C07270=1013.905,188.212,370.193,167.076,55.174,160.197
C07271=1013.901,187.964,370.214,167.071,55.186,160.199
C07272=1013.897,187.715,370.234,167.066,55.198,160.200
C07273=1013.892,187.466,370.256,167.063,55.210,160.202
C07274=1013.889,187.217,370.278,167.058,55.222,160.203
C07275=1013.885,186.938,370.301,167.053,55.235,160.205
C07276=1013.881,186.658,370.325,167.049,55.249,160.206
C07277=1013.875,186.380,370.348,167.043,55.262,160.208
C07278=1013.871,186.100,370.372,167.039,55.275,160.209
C07279=1013.867,185.851,370.393,167.035,55.287,160.211
C07280=1013.863,185.602,370.414,167.030,55.299,160.212
C07281=1013.859,185.352,370.435,167.026,55.311,160.214
C07282=1013.855,185.104,370.456,167.023,55.323,160.215
C07283=1013.852,184.855,370.477,167.018,55.335,160.217
C07284=1013.847,184.605,370.499,167.013,55.347,160.218
C07285=1013.843,184.356,370.519,167.010,55.358,160.220
C07286=1013.839,184.108,370.540,167.005,55.370,160.221
C07287=1013.836,183.858,370.562,167.001,55.382,160.222
C07288=1013.832,183.609,370.583,166.997,55.393,160.224
C07289=1013.828,183.360,370.603,166.993,55.406,160.225
C07290=1013.824,183.110,370.624,166.989,55.418,160.227
C07291=1013.820,182.861,370.645,166.985,55.430,160.228
C07292=1013.817,182.613,370.666,166.980,55.441,160.230
C07293=1013.813,182.364,370.687,166.976,55.453,160.231
C07294=1013.809,182.114,370.708,166.972,55.465,160.233
C07295=1013.805,181.865,370.729,166.968,55.476,160.234
C07296=1013.801,181.615,370.750,166.964,55.488,160.235
C07297=1013.797,181.367,370.770,166.960,55.501,160.237
C07298=1013.793,181.118,370.791,166.956,55.512,160.239
C07299=1013.788,180.868,370.811,166.951,55.524,160.240
C07300=1013.784,180.619,370.832,166.947,55.537,160.241
C07301=1013.780,180.370,370.852,166.943,55.549,160.243
C07302=1013.776,180.122,370.872,166.939,55.561,160.244
C07303=1013.772,179.872,370.893,166.935,55.573,160.246
C07304=1013.767,179.623,370.912,166.931,55.585,160.247
C07305=1013.763,179.374,370.933,166.927,55.598,160.249
C07306=1013.760,179.124,370.953,166.923,55.609,160.250
C07307=1013.754,178.875,370.973,166.918,55.621,160.252
C07308=1013.751,178.626,370.994,166.914,55.634,160.253
C07309=1013.746,178.377,371.013,166.911,55.645,160.255
C07310=1013.743,178.128,371.034,166.906,55.657,160.256
C07311=1013.738,177.878,371.054,166.902,55.670,160.258
C07312=1013.734,177.630,371.074,166.898,55.682,160.259
C07313=1013.730,177.380,371.094,166.894,55.694,160.261
C07314=1013.726,177.131,371.114,166.890,55.706,160.262
C07315=1013.721,176.882,371.135,166.886,55.718,160.264
C07316=1013.718,176.633,371.155,166.882,55.730,160.265
C07317=1013.713,176.384,371.175,166.878,55.743,160.267
C07318=1013.709,176.135,371.195,166.875,55.754,160.268
C07319=1013.705,175.886,371.215,166.870,55.766,160.270
C07320=1013.701,175.636,371.235,166.866,55.778,160.271
C07321=1013.697,175.387,371.256,166.863,55.790,160.273
C07322=1013.693,175.138,371.276,166.858,55.802,160.274
C07323=1013.689,174.889,371.296,166.854,55.814,160.276
C07324=1013.685,174.640,371.315,166.851,55.827,160.278
C07325=1013.681,174.391,371.336,166.846,55.839,160.279
C07326=1013.677,174.141,371.356,166.843,55.850,160.280
C07327=1013.673,173.892,371.375,166.838,55.862,160.282
C07328=1013.668,173.642,371.396,166.835,55.875,160.284
C07329=1013.664,173.394,371.416,166.831,55.887,160.285
C07330=1013.660,173.145,371.436,166.826,55.899,160.286
C07331=1013.657,172.895,371.456,166.823,55.910,160.288
C07332=1013.652,172.646,371.476,166.819,55.923,160.289
C07333=1013.648,172.397,371.496,166.816,55.935,160.291
C07334=1013.644,172.148,371.516,166.811,55.947,160.292
C07335=1013.640,171.899,371.536,166.808,55.958,160.294
C07336=1013.636,171.650,371.555,166.803,55.970,160.295
C07337=1013.632,171.401,371.576,166.800,55.983,160.297
C07338=1013.629,171.151,371.596,166.796,55.995,160.298
C07339=1013.624,170.872,371.619,166.792,56.007,160.300
C07340=1013.619,170.593,371.641,166.787,56.021,160.302
C07341=1013.615,170.314,371.663,166.784,56.034,160.303
C07342=1013.610,170.034,371.685,166.779,56.048,160.305
C07343=1013.606,169.785,371.705,166.775,56.060,160.307
C07344=1013.603,169.536,371.725,166.771,56.072,160.308
C07345=1013.598,169.287,371.745,166.768,56.083,160.310
C07346=1013.595,169.037,371.765,166.763,56.095,160.311
C07347=1013.591,168.788,371.784,166.761,56.108,160.313
C07348=1013.587,168.539,371.804,166.756,56.120,160.314
C07349=1013.583,168.290,371.824,166.753,56.131,160.316
C07350=1013.579,168.041,371.845,166.749,56.143,160.317
C07351=1013.575,167.792,371.865,166.745,56.155,160.319
C07352=1013.571,167.543,371.884,166.742,56.167,160.320
C07353=1013.567,167.293,371.904,166.737,56.179,160.322
C07354=1013.563,167.044,371.924,166.734,56.190,160.323
C07355=1013.559,166.795,371.944,166.730,56.202,160.325
C07356=1013.556,166.546,371.964,166.726,56.214,160.326
C07357=1013.551,166.297,371.983,166.723,56.227,160.328
C07358=1013.548,166.047,372.003,166.720,56.238,160.329
C07359=1013.543,165.798,372.023,166.715,56.250,160.331
C07360=1013.540,165.549,372.043,166.712,56.262,160.332
C07361=1013.535,165.300,372.062,166.709,56.274,160.334
C07362=1013.532,165.050,372.082,166.704,56.286,160.335
C07363=1013.528,164.801,372.102,166.701,56.297,160.337
C07364=1013.524,164.552,372.122,166.698,56.309,160.338
C07365=1013.521,164.303,372.142,166.694,56.321,160.340
C07366=1013.517,164.054,372.160,166.690,56.333,160.341
C07367=1013.513,163.804,372.180,166.687,56.345,160.343
C07368=1013.509,163.555,372.200,166.683,56.356,160.344
C07369=1013.505,163.306,372.220,166.680,56.368,160.346
C07370=1013.501,163.057,372.240,166.676,56.380,160.347
C07371=1013.497,162.808,372.259,166.672,56.392,160.349
C07372=1013.493,162.558,372.280,166.669,56.403,160.350
C07373=1013.490,162.310,372.299,166.666,56.415,160.352
C07374=1013.486,162.061,372.319,166.661,56.427,160.353
C07375=1013.482,161.812,372.338,166.658,56.439,160.355
C07376=1013.478,161.562,372.358,166.654,56.450,160.356
C07377=1013.475,161.312,372.378,166.651,56.462,160.358
C07378=1013.471,161.063,372.397,166.648,56.473,160.359
C07379=1013.467,160.814,372.417,166.644,56.485,160.361
C07380=1013.463,160.565,372.436,166.640,56.497,160.362
C07381=1013.460,160.316,372.456,166.637,56.509,160.364
C07382=1013.456,160.066,372.476,166.633,56.521,160.365
C07383=1013.452,159.817,372.495,166.630,56.532,160.367
C07384=1013.448,159.568,372.515,166.627,56.544,160.368
C07385=1013.445,159.319,372.534,166.624,56.556,160.370
C07386=1013.441,159.070,372.554,166.620,56.567,160.371
C07387=1013.437,158.820,372.573,166.616,56.579,160.373
C07388=1013.433,158.571,372.593,166.612,56.591,160.374
C07389=1013.430,158.322,372.613,166.609,56.603,160.376
C07390=1013.426,158.072,372.632,166.606,56.614,160.377
C07391=1013.421,157.823,372.652,166.603,56.626,160.379
C07392=1013.418,157.574,372.670,166.599,56.638,160.381
C07393=1013.413,157.325,372.689,166.595,56.650,160.382
C07394=1013.410,157.075,372.709,166.592,56.662,160.384
C07395=1013.406,156.826,372.728,166.589,56.673,160.385
C07396=1013.402,156.577,372.747,166.585,56.685,160.387
C07397=1013.398,156.328,372.766,166.582,56.697,160.388
C07398=1013.394,156.078,372.785,166.578,56.709,160.390
C07399=1013.390,155.829,372.804,166.575,56.721,160.391
C07400=1013.386,155.580,372.823,166.571,56.733,160.393
C07401=1013.382,155.331,372.842,166.568,56.744,160.394
C07402=1013.378,155.082,372.861,166.565,56.756,160.396
C07403=1013.374,154.802,372.882,166.560,56.769,160.397
C07404=1013.370,154.522,372.904,166.557,56.783,160.399
C07405=1013.365,154.243,372.925,166.553,56.796,160.401
C07406=1013.360,153.963,372.947,166.550,56.809,160.403
C07407=1013.357,153.714,372.965,166.547,56.821,160.404
C07408=1013.352,153.465,372.984,166.542,56.833,160.406
C07409=1013.348,153.216,373.003,166.539,56.845,160.407
C07410=1013.344,152.966,373.022,166.536,56.857,160.409
C07411=1013.341,152.718,373.041,166.533,56.868,160.411
C07412=1013.337,152.468,373.060,166.530,56.880,160.412
C07413=1013.333,152.218,373.079,166.526,56.891,160.413
C07414=1013.329,151.970,373.098,166.523,56.903,160.415
C07415=1013.325,151.720,373.116,166.520,56.915,160.417
C07416=1013.321,151.471,373.135,166.516,56.927,160.418
C07417=1013.317,151.222,373.154,166.513,56.938,160.420
C07418=1013.313,150.972,373.172,166.510,56.950,160.421
C07419=1013.309,150.723,373.192,166.507,56.962,160.423
C07420=1013.305,150.474,373.210,166.503,56.974,160.424
C07421=1013.301,150.224,373.229,166.500,56.986,160.426
C07422=1013.297,149.975,373.248,166.497,56.998,160.427
C07423=1013.293,149.726,373.267,166.493,57.009,160.429
C07424=1013.289,149.477,373.286,166.490,57.021,160.430
C07425=1013.285,149.227,373.304,166.487,57.033,160.432
C07426=1013.282,148.978,373.323,166.483,57.044,160.434
C07427=1013.278,148.728,373.341,166.480,57.056,160.435
C07428=1013.274,148.479,373.360,166.477,57.068,160.437
C07429=1013.270,148.230,373.379,166.474,57.079,160.438
C07430=1013.266,147.981,373.398,166.470,57.091,160.440
C07431=1013.262,147.732,373.416,166.467,57.103,160.441
C07432=1013.258,147.482,373.435,166.464,57.115,160.443
C07433=1013.254,147.233,373.453,166.461,57.126,160.444
C07434=1013.250,146.984,373.472,166.457,57.138,160.446
C07435=1013.246,146.734,373.491,166.454,57.149,160.447
C07436=1013.243,146.485,373.509,166.451,57.161,160.449
C07437=1013.239,146.235,373.528,166.449,57.173,160.451
C07438=1013.235,145.987,373.545,166.446,57.184,160.452
C07439=1013.231,145.737,373.564,166.442,57.196,160.454
C07440=1013.227,145.487,373.583,166.439,57.207,160.455
C07441=1013.223,145.239,373.602,166.436,57.219,160.457
C07442=1013.219,144.989,373.621,166.433,57.231,160.458
C07443=1013.215,144.740,373.638,166.430,57.242,160.460
C07444=1013.211,144.491,373.657,166.427,57.254,160.461
C07445=1013.207,144.242,373.675,166.424,57.266,160.463
C07446=1013.203,143.992,373.693,166.420,57.278,160.465
C07447=1013.199,143.743,373.712,166.417,57.290,160.466
C07448=1013.195,143.494,373.730,166.414,57.301,160.468
C07449=1013.191,143.245,373.748,166.411,57.313,160.469
C07450=1013.187,142.995,373.767,166.408,57.325,160.471
C07451=1013.183,142.746,373.786,166.405,57.336,160.472
C07452=1013.179,142.496,373.803,166.402,57.347,160.474
C07453=1013.175,142.247,373.822,166.399,57.359,160.475
C07454=1013.172,141.998,373.840,166.396,57.371,160.477
C07455=1013.167,141.748,373.858,166.392,57.382,160.478
C07456=1013.163,141.499,373.876,166.389,57.394,160.480
C07457=1013.159,141.250,373.895,166.386,57.406,160.482
C07458=1013.155,141.000,373.912,166.383,57.417,160.483
C07459=1013.152,140.752,373.931,166.381,57.428,160.485
C07460=1013.148,140.502,373.949,166.378,57.440,160.486
C07461=1013.144,140.253,373.967,166.374,57.452,160.488
C07462=1013.140,140.004,373.986,166.371,57.463,160.489
C07463=1013.136,139.754,374.003,166.368,57.475,160.491
C07464=1013.132,139.505,374.022,166.366,57.486,160.492
C07465=1013.128,139.256,374.040,166.363,57.498,160.494
C07466=1013.124,139.006,374.058,166.359,57.509,160.495
C07467=1013.120,138.726,374.079,166.356,57.522,160.497
C07468=1013.115,138.447,374.100,166.352,57.535,160.499
C07469=1013.111,138.167,374.119,166.350,57.548,160.501
C07470=1013.107,137.888,374.140,166.347,57.561,160.503
C07471=1013.103,137.639,374.158,166.343,57.572,160.504
C07472=1013.099,137.389,374.176,166.340,57.584,160.506
C07473=1013.095,137.140,374.194,166.338,57.595,160.507
C07474=1013.090,136.891,374.212,166.335,57.607,160.509
C07475=1013.087,136.641,374.230,166.332,57.619,160.510
C07476=1013.083,136.393,374.248,166.328,57.630,160.512
C07477=1013.079,136.142,374.266,166.326,57.641,160.513
C07478=1013.075,135.894,374.284,166.323,57.653,160.515
C07479=1013.071,135.644,374.302,166.320,57.665,160.516
C07480=1013.067,135.395,374.320,166.316,57.676,160.518
C07481=1013.064,135.146,374.338,166.314,57.687,160.520
C07482=1013.059,134.896,374.355,166.311,57.698,160.521
C07483=1013.055,134.647,374.373,166.308,57.710,160.523
C07484=1013.051,134.397,374.391,166.305,57.721,160.524
C07485=1013.047,134.148,374.409,166.302,57.733,160.526
C07486=1013.044,133.899,374.427,166.299,57.744,160.527
C07487=1013.039,133.649,374.445,166.297,57.756,160.529
C07488=1013.035,133.400,374.462,166.294,57.767,160.530
C07489=1013.032,133.151,374.480,166.291,57.779,160.532
C07490=1013.028,132.901,374.498,166.288,57.790,160.533
C07491=1013.023,132.653,374.516,166.285,57.802,160.535
C07492=1013.020,132.403,374.533,166.282,57.813,160.536
C07493=1013.015,132.154,374.551,166.279,57.824,160.538
C07494=1013.012,131.904,374.569,166.277,57.836,160.540
C07495=1013.008,131.655,374.587,166.274,57.847,160.541
C07496=1013.004,131.405,374.604,166.271,57.859,160.543
C07497=1013.001,131.156,374.622,166.268,57.870,160.544
C07498=1012.996,130.907,374.640,166.265,57.881,160.546
C07499=1012.992,130.657,374.657,166.263,57.893,160.547
C07500=1012.988,130.408,374.676,166.260,57.903,160.549
C07501=1012.985,130.159,374.693,166.257,57.915,160.550
C07502=1012.981,129.909,374.711,166.255,57.926,160.552
C07503=1012.977,129.660,374.729,166.251,57.937,160.553
C07504=1012.973,129.411,374.746,166.249,57.948,160.555
C07505=1012.969,129.161,374.764,166.246,57.960,160.557
C07506=1012.965,128.912,374.781,166.243,57.972,160.558
C07507=1012.961,128.663,374.799,166.240,57.982,160.559
C07508=1012.957,128.413,374.816,166.237,57.994,160.561
C07509=1012.953,128.163,374.833,166.235,58.005,160.563
C07510=1012.949,127.914,374.850,166.232,58.017,160.564
C07511=1012.945,127.665,374.868,166.229,58.028,160.566
C07512=1012.940,127.415,374.885,166.226,58.039,160.567
C07513=1012.936,127.166,374.902,166.224,58.051,160.569
C07514=1012.932,126.917,374.920,166.221,58.062,160.570
C07515=1012.928,126.667,374.937,166.218,58.073,160.572
C07516=1012.924,126.418,374.954,166.216,58.085,160.574
C07517=1012.920,126.168,374.971,166.213,58.096,160.575
C07518=1012.916,125.920,374.989,166.210,58.107,160.577
C07519=1012.911,125.670,375.006,166.208,58.119,160.578
C07520=1012.908,125.420,375.023,166.205,58.130,160.580
C07521=1012.904,125.171,375.041,166.202,58.141,160.581
C07522=1012.900,124.922,375.058,166.199,58.152,160.583
C07523=1012.896,124.673,375.075,166.197,58.164,160.584
C07524=1012.892,124.423,375.092,166.194,58.175,160.586
C07525=1012.888,124.173,375.109,166.191,58.186,160.587
C07526=1012.884,123.924,375.126,166.189,58.197,160.589
C07527=1012.880,123.675,375.143,166.186,58.208,160.591
C07528=1012.876,123.426,375.161,166.184,58.220,160.592
C07529=1012.871,123.176,375.179,166.181,58.231,160.594
C07530=1012.867,122.927,375.196,166.178,58.242,160.595
C07531=1012.863,122.621,375.216,166.175,58.255,160.597
C07532=1012.858,122.316,375.237,166.172,58.269,160.599
C07533=1012.853,122.010,375.258,166.169,58.282,160.601
C07534=1012.849,121.705,375.280,166.165,58.296,160.602
C07535=1012.844,121.455,375.297,166.162,58.307,160.604
C07536=1012.840,121.206,375.314,166.160,58.318,160.606
C07537=1012.836,120.956,375.331,166.158,58.330,160.607
C07538=1012.832,120.707,375.348,166.155,58.341,160.609
C07539=1012.829,120.458,375.366,166.153,58.352,160.610
C07540=1012.825,120.208,375.383,166.151,58.363,160.612
C07541=1012.820,119.959,375.400,166.147,58.374,160.613
C07542=1012.816,119.709,375.417,166.145,58.385,160.615
C07543=1012.813,119.460,375.434,166.142,58.395,160.616
C07544=1012.809,119.211,375.451,166.140,58.406,160.618
C07545=1012.805,118.961,375.468,166.136,58.417,160.619
C07546=1012.801,118.712,375.485,166.134,58.428,160.621
C07547=1012.797,118.463,375.503,166.132,58.439,160.622
C07548=1012.793,118.214,375.520,166.130,58.450,160.624
C07549=1012.789,117.964,375.537,166.127,58.461,160.626
C07550=1012.785,117.714,375.554,166.124,58.472,160.627
C07551=1012.781,117.465,375.571,166.122,58.483,160.628
C07552=1012.777,117.216,375.588,166.120,58.494,160.630
C07553=1012.773,116.966,375.605,166.117,58.504,160.631
C07554=1012.770,116.717,375.622,166.115,58.515,160.633
C07555=1012.766,116.467,375.639,166.112,58.526,160.635
C07556=1012.762,116.218,375.656,166.110,58.537,160.636
C07557=1012.758,115.969,375.673,166.108,58.548,160.638
C07558=1012.754,115.720,375.690,166.104,58.558,160.639
C07559=1012.750,115.470,375.707,166.102,58.569,160.640
C07560=1012.746,115.221,375.724,166.099,58.580,160.642
C07561=1012.742,114.971,375.742,166.097,58.591,160.644
C07562=1012.738,114.722,375.759,166.094,58.601,160.645
C07563=1012.734,114.472,375.775,166.092,58.612,160.646
C07564=1012.731,114.223,375.792,166.090,58.623,160.648
C07565=1012.727,113.973,375.809,166.087,58.633,160.649
C07566=1012.723,113.724,375.826,166.085,58.644,160.651
C07567=1012.719,113.475,375.843,166.083,58.655,160.652
C07568=1012.715,113.226,375.860,166.080,58.665,160.654
C07569=1012.711,112.976,375.878,166.078,58.676,160.655
C07570=1012.708,112.726,375.894,166.076,58.687,160.657
C07571=1012.704,112.477,375.911,166.073,58.697,160.658
C07572=1012.700,112.228,375.928,166.071,58.708,160.660
C07573=1012.696,111.979,375.945,166.068,58.719,160.661
C07574=1012.692,111.729,375.962,166.066,58.729,160.663
C07575=1012.689,111.479,375.979,166.063,58.740,160.664
C07576=1012.685,111.230,375.996,166.061,58.751,160.666
C07577=1012.680,110.981,376.012,166.059,58.762,160.667
C07578=1012.677,110.731,376.029,166.056,58.772,160.669
C07579=1012.673,110.482,376.046,166.054,58.783,160.670
C07580=1012.669,110.233,376.063,166.051,58.794,160.672
C07581=1012.664,109.983,376.078,166.050,58.803,160.673
C07582=1012.661,109.734,376.096,166.048,58.814,160.675
C07583=1012.657,109.484,376.112,166.045,58.825,160.676
C07584=1012.652,109.235,376.128,166.043,58.836,160.678
C07585=1012.649,108.986,376.145,166.040,58.846,160.679
C07586=1012.645,108.736,376.162,166.038,58.857,160.681
C07587=1012.611,121.701,374.880,166.126,58.488,160.631
C07588=1012.616,121.999,374.859,166.130,58.476,160.629
C07589=1012.621,122.296,374.839,166.133,58.462,160.627
C07590=1012.625,122.594,374.819,166.135,58.450,160.625
C07591=1012.629,122.892,374.799,166.138,58.436,160.624
C07592=1012.634,123.142,374.781,166.142,58.425,160.622
C07593=1012.638,123.391,374.764,166.144,58.414,160.621
C07594=1012.642,123.640,374.747,166.146,58.403,160.619
C07595=1012.646,123.890,374.730,166.148,58.392,160.617
C07596=1012.649,124.139,374.713,166.152,58.381,160.616
C07597=1012.653,124.388,374.696,166.154,58.370,160.615
C07598=1012.657,124.637,374.679,166.157,58.359,160.613
C07599=1012.662,124.887,374.661,166.160,58.348,160.612
C07600=1012.666,125.137,374.644,166.162,58.337,160.610
C07601=1012.669,125.386,374.627,166.165,58.326,160.609
C07602=1012.673,125.635,374.610,166.167,58.314,160.607
C07603=1012.677,125.884,374.593,166.169,58.303,160.605
C07604=1012.682,126.134,374.575,166.173,58.292,160.604
C07605=1012.686,126.383,374.558,166.175,58.281,160.602
C07606=1012.690,126.632,374.541,166.178,58.270,160.601
C07607=1012.694,126.882,374.523,166.181,58.259,160.599
C07608=1012.697,127.131,374.506,166.183,58.247,160.598
C07609=1012.702,127.381,374.489,166.186,58.236,160.596
C07610=1012.706,127.630,374.472,166.189,58.225,160.595
C07611=1012.710,127.879,374.455,166.191,58.214,160.593
C07612=1012.714,128.129,374.438,166.195,58.202,160.592
C07613=1012.717,128.378,374.421,166.196,58.191,160.590
C07614=1012.722,128.628,374.403,166.200,58.180,160.588
C07615=1012.726,128.877,374.386,166.202,58.169,160.587
C07616=1012.730,129.126,374.369,166.205,58.157,160.586
C07617=1012.734,129.375,374.351,166.207,58.146,160.584
C07618=1012.738,129.625,374.333,166.211,58.135,160.582
C07619=1012.741,129.875,374.316,166.213,58.124,160.581
C07620=1012.745,130.124,374.298,166.216,58.112,160.579
C07621=1012.749,130.373,374.281,166.219,58.102,160.578
C07622=1012.753,130.623,374.263,166.222,58.090,160.576
C07623=1012.757,130.872,374.245,166.224,58.079,160.575
C07624=1012.760,131.121,374.228,166.227,58.067,160.573
C07625=1012.764,131.371,374.210,166.230,58.057,160.572
C07626=1012.768,131.620,374.192,166.232,58.045,160.570
C07627=1012.772,131.869,374.175,166.235,58.034,160.568
C07628=1012.775,132.119,374.157,166.238,58.023,160.567
C07629=1012.780,132.368,374.139,166.241,58.012,160.566
C07630=1012.784,132.617,374.122,166.243,58.000,160.564
C07631=1012.788,132.866,374.104,166.246,57.989,160.562
C07632=1012.791,133.116,374.086,166.249,57.978,160.561
C07633=1012.795,133.366,374.068,166.252,57.966,160.559
C07634=1012.799,133.615,374.051,166.255,57.955,160.558
C07635=1012.803,133.864,374.034,166.258,57.944,160.556
C07636=1012.807,134.114,374.015,166.260,57.932,160.555
C07637=1012.811,134.363,373.998,166.263,57.921,160.553
C07638=1012.815,134.612,373.981,166.266,57.909,160.552
C07639=1012.819,134.862,373.962,166.268,57.898,160.550
C07640=1012.823,135.111,373.945,166.272,57.887,160.549
C07641=1012.826,135.360,373.926,166.275,57.875,160.547
C07642=1012.831,135.610,373.909,166.277,57.864,160.546
C07643=1012.834,135.859,373.891,166.280,57.852,160.544
C07644=1012.838,136.108,373.873,166.284,57.841,160.543
C07645=1012.842,136.358,373.855,166.285,57.829,160.541
C07646=1012.846,136.607,373.838,166.289,57.818,160.539
C07647=1012.849,136.856,373.819,166.292,57.807,160.538
C07648=1012.854,137.105,373.801,166.294,57.795,160.536
C07649=1012.857,137.355,373.783,166.298,57.784,160.535
C07650=1012.862,137.604,373.766,166.301,57.772,160.533
C07651=1012.865,137.854,373.748,166.303,57.761,160.532
C07652=1012.870,138.133,373.727,166.306,57.748,160.530
C07653=1012.874,138.413,373.707,166.310,57.735,160.528
C07654=1012.878,138.691,373.687,166.314,57.723,160.527
C07655=1012.882,138.971,373.667,166.316,57.710,160.525
C07656=1012.887,139.221,373.648,166.319,57.698,160.523
C07657=1012.890,139.470,373.630,166.322,57.687,160.522
C07658=1012.894,139.719,373.613,166.325,57.675,160.520
C07659=1012.898,139.969,373.594,166.328,57.664,160.519
C07660=1012.902,140.217,373.576,166.331,57.652,160.517
C07661=1012.906,140.467,373.557,166.334,57.641,160.516
C07662=1012.909,140.717,373.540,166.337,57.629,160.514
C07663=1012.914,140.966,373.522,166.341,57.618,160.513
C07664=1012.917,141.215,373.503,166.343,57.606,160.511
C07665=1012.921,141.464,373.485,166.346,57.594,160.509
C07666=1012.925,141.714,373.467,166.349,57.583,160.508
C07667=1012.929,141.963,373.449,166.352,57.571,160.506
C07668=1012.933,142.212,373.430,166.356,57.560,160.505
C07669=1012.937,142.461,373.412,166.359,57.548,160.503
C07670=1012.941,142.711,373.394,166.361,57.537,160.501
C07671=1012.944,142.960,373.376,166.364,57.526,160.500
C07672=1012.949,143.210,373.358,166.367,57.514,160.498
C07673=1012.952,143.459,373.339,166.370,57.502,160.497
C07674=1012.956,143.708,373.321,166.374,57.491,160.496
C07675=1012.960,143.958,373.304,166.377,57.479,160.494
C07676=1012.964,144.206,373.285,166.380,57.467,160.492
C07677=1012.968,144.456,373.266,166.383,57.455,160.491
C07678=1012.972,144.705,373.249,166.386,57.444,160.489
C07679=1012.976,144.954,373.230,166.389,57.432,160.488
C07680=1012.979,145.203,373.211,166.392,57.420,160.486
C07681=1012.984,145.453,373.193,166.395,57.409,160.485
C07682=1012.987,145.702,373.176,166.398,57.397,160.483
C07683=1012.991,145.952,373.157,166.401,57.385,160.481
C07684=1012.995,146.202,373.138,166.404,57.374,160.480
C07685=1012.999,146.451,373.120,166.407,57.362,160.478
C07686=1013.003,146.700,373.101,166.410,57.351,160.477
C07687=1013.006,146.949,373.083,166.414,57.339,160.475
C07688=1013.010,147.199,373.064,166.417,57.327,160.474
C07689=1013.015,147.448,373.046,166.420,57.316,160.472
C07690=1013.019,147.697,373.027,166.423,57.304,160.471
C07691=1013.022,147.946,373.009,166.426,57.292,160.469
C07692=1013.026,148.196,372.990,166.430,57.281,160.468
C07693=1013.030,148.444,372.971,166.433,57.269,160.466
C07694=1013.034,148.694,372.952,166.436,57.257,160.464
C07695=1013.038,148.943,372.934,166.439,57.245,160.463
C07696=1013.041,149.192,372.915,166.443,57.234,160.462
C07697=1013.045,149.442,372.896,166.446,57.222,160.460
C07698=1013.049,149.691,372.878,166.449,57.210,160.458
C07699=1013.053,149.941,372.859,166.452,57.198,160.457
C07700=1013.056,150.190,372.841,166.455,57.187,160.455
C07701=1013.060,150.439,372.822,166.459,57.176,160.454
C07702=1013.065,150.688,372.803,166.462,57.164,160.452
C07703=1013.069,150.937,372.785,166.465,57.152,160.451
C07704=1013.073,151.187,372.766,166.468,57.140,160.449
C07705=1013.076,151.436,372.748,166.471,57.128,160.447
C07706=1013.081,151.685,372.729,166.474,57.116,160.446
C07707=1013.085,151.935,372.710,166.477,57.104,160.444
C07708=1013.088,152.184,372.692,166.482,57.093,160.443
C07709=1013.092,152.433,372.672,166.485,57.081,160.441
C07710=1013.096,152.683,372.654,166.488,57.069,160.440
C07711=1013.100,152.932,372.635,166.491,57.057,160.438
C07712=1013.104,153.181,372.616,166.494,57.046,160.437
C07713=1013.107,153.430,372.597,166.497,57.034,160.435
C07714=1013.111,153.680,372.578,166.501,57.022,160.434
C07715=1013.115,153.929,372.559,166.504,57.011,160.432
C07716=1013.120,154.208,372.538,166.507,56.997,160.430
C07717=1013.124,154.487,372.517,166.512,56.984,160.429
C07718=1013.128,154.767,372.495,166.516,56.971,160.427
C07719=1013.133,155.047,372.474,166.519,56.958,160.425
C07720=1013.137,155.295,372.455,166.522,56.946,160.424
C07721=1013.141,155.545,372.437,166.527,56.934,160.422
C07722=1013.144,155.795,372.417,166.530,56.922,160.421
C07723=1013.148,156.043,372.398,166.533,56.910,160.419
C07724=1013.152,156.293,372.379,166.536,56.899,160.418
C07725=1013.156,156.542,372.361,166.539,56.887,160.416
C07726=1013.160,156.791,372.341,166.543,56.875,160.415
C07727=1013.163,157.040,372.323,166.547,56.863,160.413
C07728=1013.168,157.289,372.303,166.550,56.851,160.411
C07729=1013.172,157.539,372.285,166.553,56.839,160.410
C07730=1013.175,157.788,372.266,166.557,56.827,160.408
C07731=1013.180,158.037,372.247,166.560,56.815,160.407
C07732=1013.183,158.287,372.227,166.563,56.803,160.405
C07733=1013.187,158.536,372.208,166.567,56.792,160.404
C07734=1013.191,158.785,372.188,166.570,56.780,160.402
C07735=1013.194,159.035,372.169,166.573,56.768,160.400
C07736=1013.198,159.284,372.149,166.577,56.757,160.399
C07737=1013.202,159.533,372.129,166.581,56.745,160.398
C07738=1013.206,159.783,372.110,166.584,56.733,160.396
C07739=1013.209,160.031,372.091,166.588,56.721,160.395
C07740=1013.212,160.281,372.071,166.591,56.710,160.393
C07741=1013.217,160.530,372.051,166.594,56.698,160.391
C07742=1013.220,160.780,372.032,166.597,56.686,160.390
C07743=1013.224,161.028,372.013,166.601,56.674,160.389
C07744=1013.227,161.277,371.993,166.605,56.662,160.387
C07745=1013.232,161.526,371.973,166.608,56.651,160.386
C07746=1013.235,161.776,371.954,166.612,56.639,160.384
C07747=1013.239,162.026,371.934,166.615,56.628,160.383
C07748=1013.242,162.274,371.915,166.619,56.615,160.381
C07749=1013.246,162.523,371.895,166.622,56.604,160.380
C07750=1013.250,162.772,371.875,166.626,56.592,160.378
C07751=1013.254,163.022,371.856,166.629,56.580,160.376
C07752=1013.258,163.271,371.836,166.633,56.568,160.375
C07753=1013.261,163.520,371.817,166.637,56.556,160.373
C07754=1013.265,163.769,371.797,166.640,56.545,160.372
C07755=1013.269,164.019,371.777,166.644,56.533,160.371
C07756=1013.272,164.268,371.757,166.647,56.521,160.369
C07757=1013.277,164.517,371.738,166.651,56.509,160.367
C07758=1013.280,164.767,371.718,166.655,56.497,160.366
C07759=1013.283,165.016,371.699,166.658,56.485,160.364
C07760=1013.287,165.265,371.679,166.662,56.473,160.363
C07761=1013.291,165.514,371.659,166.666,56.461,160.361
C07762=1013.295,165.763,371.640,166.669,56.450,160.360
C07763=1013.299,166.012,371.619,166.672,56.438,160.358
C07764=1013.303,166.261,371.600,166.677,56.426,160.357
C07765=1013.307,166.511,371.580,166.680,56.414,160.355
C07766=1013.311,166.760,371.560,166.683,56.402,160.354
C07767=1013.315,167.009,371.540,166.687,56.390,160.352
C07768=1013.318,167.258,371.521,166.690,56.378,160.351
C07769=1013.322,167.507,371.502,166.695,56.366,160.349
C07770=1013.326,167.757,371.482,166.698,56.354,160.348
C07771=1013.329,168.006,371.462,166.701,56.342,160.346
C07772=1013.334,168.255,371.442,166.706,56.330,160.345
C07773=1013.337,168.505,371.422,166.709,56.319,160.343
C07774=1013.342,168.754,371.403,166.714,56.307,160.342
C07775=1013.345,169.003,371.383,166.716,56.294,160.340
C07776=1013.349,169.252,371.363,166.721,56.282,160.339
C07777=1013.353,169.501,371.343,166.724,56.270,160.337
C07778=1013.357,169.751,371.323,166.728,56.258,160.336
C07779=1013.361,170.000,371.304,166.732,56.247,160.334
C07780=1013.366,170.278,371.281,166.736,56.233,160.332
C07781=1013.370,170.557,371.259,166.740,56.220,160.331
C07782=1013.374,170.837,371.236,166.744,56.206,160.329
C07783=1013.379,171.116,371.214,166.749,56.193,160.327
C07784=1013.383,171.365,371.194,166.752,56.180,160.326
C07785=1013.386,171.615,371.174,166.756,56.168,160.324
C07786=1013.391,171.864,371.155,166.760,56.157,160.323
C07787=1013.394,172.113,371.135,166.764,56.145,160.321
C07788=1013.398,172.362,371.115,166.768,56.133,160.320
C07789=1013.402,172.611,371.095,166.772,56.120,160.318
C07790=1013.406,172.861,371.075,166.776,56.108,160.317
C07791=1013.411,173.109,371.055,166.779,56.096,160.315
C07792=1013.414,173.359,371.035,166.784,56.084,160.314
C07793=1013.418,173.608,371.015,166.787,56.072,160.312
C07794=1013.422,173.857,370.995,166.791,56.060,160.311
C07795=1013.426,174.106,370.975,166.796,56.048,160.309
C07796=1013.430,174.355,370.956,166.798,56.036,160.307
C07797=1013.434,174.604,370.935,166.803,56.024,160.306
C07798=1013.438,174.853,370.915,166.807,56.011,160.305
C07799=1013.443,175.103,370.895,166.811,56.000,160.303
C07800=1013.446,175.352,370.875,166.815,55.987,160.302
C07801=1013.451,175.602,370.856,166.818,55.976,160.300
C07802=1013.455,175.850,370.835,166.823,55.963,160.299
C07803=1013.458,176.100,370.815,166.826,55.951,160.297
C07804=1013.462,176.349,370.795,166.831,55.939,160.296
C07805=1013.466,176.598,370.775,166.834,55.927,160.294
C07806=1013.471,176.846,370.755,166.838,55.914,160.292
C07807=1013.474,177.096,370.735,166.843,55.902,160.291
C07808=1013.479,177.346,370.715,166.846,55.891,160.290
C07809=1013.483,177.595,370.695,166.850,55.878,160.288
C07810=1013.487,177.844,370.674,166.855,55.866,160.287
C07811=1013.491,178.093,370.655,166.859,55.853,160.285
C07812=1013.495,178.342,370.635,166.862,55.842,160.283
C07813=1013.499,178.590,370.615,166.867,55.830,160.282
C07814=1013.504,178.840,370.594,166.871,55.817,160.280
C07815=1013.507,179.090,370.574,166.875,55.805,160.279
C07816=1013.512,179.338,370.554,166.879,55.793,160.277
C07817=1013.516,179.588,370.534,166.883,55.781,160.276
C07818=1013.520,179.837,370.514,166.887,55.769,160.274
C07819=1013.524,180.086,370.493,166.891,55.756,160.273
C07820=1013.528,180.335,370.473,166.896,55.744,160.272
C07821=1013.532,180.584,370.454,166.899,55.732,160.270
C07822=1013.536,180.833,370.433,166.903,55.720,160.268
C07823=1013.541,181.082,370.413,166.908,55.708,160.267
C07824=1013.545,181.332,370.392,166.912,55.695,160.265
C07825=1013.549,181.581,370.372,166.916,55.683,160.264
C07826=1013.552,181.830,370.351,166.920,55.672,160.262
C07827=1013.556,182.080,370.330,166.924,55.660,160.261
C07828=1013.560,182.329,370.310,166.928,55.647,160.259
C07829=1013.564,182.578,370.289,166.932,55.635,160.258
C07830=1013.567,182.827,370.267,166.936,55.623,160.257
C07831=1013.572,183.076,370.246,166.941,55.612,160.255
C07832=1013.575,183.325,370.226,166.944,55.600,160.254
C07833=1013.579,183.574,370.206,166.949,55.588,160.252
C07834=1013.582,183.823,370.184,166.953,55.575,160.251
C07835=1013.587,184.073,370.163,166.957,55.564,160.249
C07836=1013.591,184.321,370.142,166.961,55.552,160.248
C07837=1013.595,184.570,370.121,166.966,55.540,160.247
C07838=1013.598,184.819,370.100,166.969,55.528,160.245
C07839=1013.602,185.069,370.080,166.973,55.516,160.243
C07840=1013.606,185.318,370.059,166.978,55.504,160.242
C07841=1013.610,185.567,370.038,166.983,55.492,160.241
C07842=1013.614,185.816,370.016,166.986,55.480,160.239
C07843=1013.618,186.065,369.996,166.990,55.468,160.238
C07844=1013.622,186.344,369.972,166.995,55.455,160.236
C07845=1013.626,186.624,369.948,167.000,55.441,160.234
C07846=1013.631,186.903,369.925,167.005,55.428,160.233
C07847=1013.635,187.182,369.901,167.010,55.414,160.231
C07848=1013.639,187.431,369.880,167.014,55.402,160.230
C07849=1013.643,187.680,369.860,167.019,55.390,160.228
C07850=1013.647,187.929,369.838,167.022,55.378,160.227
C07851=1013.651,188.178,369.817,167.027,55.366,160.225
C07852=1013.654,188.427,369.796,167.031,55.354,160.224
C07853=1013.659,188.676,369.775,167.035,55.342,160.222
C07854=1013.663,188.925,369.754,167.040,55.330,160.221
C07855=1013.667,189.175,369.733,167.045,55.318,160.220
C07856=1013.671,189.423,369.712,167.049,55.306,160.218
C07857=1013.674,189.672,369.691,167.052,55.294,160.217
C07858=1013.679,189.921,369.669,167.057,55.282,160.215
C07859=1013.682,190.170,369.648,167.062,55.270,160.214
C07860=1013.687,190.419,369.627,167.066,55.258,160.212
C07861=1013.691,190.668,369.606,167.071,55.246,160.211
C07862=1013.695,190.918,369.584,167.075,55.234,160.210
C07863=1013.699,191.167,369.563,167.079,55.221,160.208
C07864=1013.703,191.415,369.543,167.084,55.209,160.207
C07865=1013.707,191.665,369.521,167.089,55.197,160.205
C07866=1013.710,191.914,369.500,167.093,55.185,160.204
C07867=1013.715,192.163,369.479,167.098,55.173,160.202
C07868=1013.719,192.411,369.457,167.102,55.161,160.201
C07869=1013.723,192.661,369.436,167.105,55.149,160.199
C07870=1013.727,192.910,369.415,167.110,55.137,160.198
C07871=1013.731,193.159,369.394,167.115,55.125,160.196
C07872=1013.735,193.408,369.373,167.119,55.113,160.195
C07873=1013.739,193.657,369.350,167.124,55.101,160.194
C07874=1013.743,193.906,369.330,167.128,55.089,160.192
C07875=1013.748,194.155,369.309,167.133,55.077,160.191
C07876=1013.752,194.404,369.288,167.137,55.065,160.189
C07877=1013.755,194.654,369.266,167.142,55.053,160.188
C07878=1013.760,194.903,369.244,167.146,55.040,160.186
C07879=1013.764,195.151,369.223,167.152,55.028,160.185
C07880=1013.769,195.401,369.202,167.156,55.016,160.183
C07881=1013.772,195.650,369.181,167.161,55.004,160.182
C07882=1013.777,195.899,369.159,167.166,54.992,160.181
C07883=1013.780,196.147,369.138,167.170,54.979,160.179
C07884=1013.784,196.397,369.116,167.175,54.968,160.178
C07885=1013.789,196.646,369.095,167.179,54.955,160.176
C07886=1013.793,196.895,369.074,167.184,54.943,160.175
C07887=1013.798,197.144,369.053,167.188,54.931,160.174
C07888=1013.802,197.393,369.030,167.192,54.919,160.172
C07889=1013.806,197.642,369.009,167.197,54.907,160.171
C07890=1013.810,197.891,368.988,167.201,54.895,160.169
C07891=1013.814,198.140,368.967,167.207,54.882,160.168
C07892=1013.818,198.389,368.945,167.212,54.871,160.166
C07893=1013.823,198.638,368.923,167.216,54.858,160.165
C07894=1013.827,198.887,368.902,167.221,54.846,160.164
C07895=1013.831,199.136,368.880,167.226,54.835,160.162
C07896=1013.835,199.386,368.858,167.230,54.822,160.161
C07897=1013.839,199.634,368.837,167.235,54.810,160.159
C07898=1013.843,199.884,368.815,167.240,54.799,160.158
C07899=1013.847,200.133,368.792,167.244,54.786,160.156
C07900=1013.851,200.381,368.771,167.249,54.774,160.155
C07901=1013.855,200.631,368.749,167.254,54.763,160.154
C07902=1013.859,200.880,368.727,167.258,54.751,160.152
C07903=1013.864,201.129,368.705,167.263,54.738,160.151
C07904=1013.867,201.378,368.684,167.268,54.726,160.150
C07905=1013.871,201.627,368.661,167.273,54.714,160.148
C07906=1013.876,201.876,368.639,167.278,54.703,160.147
C07907=1013.879,202.124,368.617,167.282,54.690,160.145
C07908=1013.897,203.217,368.521,167.813,54.786,160.288
C07909=1013.902,203.455,368.498,167.817,54.776,160.286
C07910=1013.907,203.693,368.476,167.821,54.765,160.285
C07911=1013.912,203.931,368.453,167.825,54.755,160.284
C07912=1013.917,204.169,368.430,167.830,54.745,160.283
C07913=1013.922,204.408,368.408,167.834,54.734,160.281
C07914=1013.927,204.646,368.384,167.838,54.723,160.280
C07915=1013.932,204.884,368.362,167.842,54.713,160.279
C07916=1013.937,205.122,368.340,167.847,54.703,160.278
C07917=1013.942,205.370,368.315,167.851,54.692,160.276
C07918=1013.947,205.620,368.292,167.856,54.681,160.275
C07919=1013.952,205.868,368.268,167.860,54.670,160.273
C07920=1013.957,206.117,368.244,167.864,54.659,160.272
C07921=1013.963,206.366,368.220,167.869,54.648,160.271
C07922=1013.968,206.615,368.196,167.874,54.638,160.270
C07923=1013.973,206.864,368.172,167.878,54.627,160.268
C07924=1013.978,207.112,368.148,167.883,54.616,160.267
C07925=1013.983,207.362,368.124,167.887,54.606,160.266
C07926=1013.989,207.610,368.100,167.891,54.595,160.264
C07927=1013.994,207.859,368.076,167.897,54.584,160.263
C07928=1013.999,208.108,368.052,167.901,54.573,160.262
C07929=1014.004,208.357,368.028,167.905,54.563,160.261
C07930=1014.009,208.605,368.004,167.909,54.552,160.259
C07931=1014.014,208.854,367.980,167.914,54.541,160.258
C07932=1014.020,209.103,367.956,167.919,54.531,160.257
C07933=1014.025,209.352,367.932,167.923,54.520,160.255
C07934=1014.030,209.600,367.907,167.927,54.510,160.254
C07935=1014.035,209.849,367.884,167.932,54.499,160.253
C07936=1014.041,210.098,367.860,167.937,54.489,160.252
C07937=1014.045,210.347,367.835,167.941,54.478,160.250
C07938=1014.050,210.595,367.811,167.945,54.468,160.249
C07939=1014.056,210.844,367.786,167.950,54.457,160.248
C07940=1014.061,211.093,367.762,167.954,54.447,160.247
C07941=1014.066,211.342,367.738,167.960,54.436,160.246
C07942=1014.071,211.591,367.714,167.964,54.426,160.244
C07943=1014.076,211.839,367.689,167.968,54.415,160.243
C07944=1014.081,212.088,367.665,167.973,54.405,160.242
C07945=1014.087,212.337,367.641,167.977,54.395,160.241
C07946=1014.091,212.585,367.616,167.981,54.384,160.239
C07947=1014.097,212.835,367.591,167.986,54.374,160.238
C07948=1014.102,213.083,367.567,167.991,54.364,160.237
C07949=1014.108,213.332,367.543,167.996,54.353,160.236
C07950=1014.113,213.580,367.519,168.000,54.343,160.235
C07951=1014.117,213.829,367.494,168.005,54.333,160.233
C07952=1014.123,214.078,367.469,168.009,54.322,160.232
C07953=1014.128,214.327,367.445,168.014,54.312,160.231
C07954=1014.133,214.575,367.421,168.018,54.302,160.230
C07955=1014.139,214.825,367.396,168.023,54.292,160.228
C07956=1014.144,215.073,367.371,168.027,54.281,160.227
C07957=1014.149,215.322,367.347,168.032,54.270,160.226
C07958=1014.154,215.570,367.323,168.037,54.261,160.225
C07959=1014.160,215.819,367.299,168.041,54.250,160.224
C07960=1014.165,216.069,367.274,168.046,54.240,160.223
C07961=1014.170,216.317,367.249,168.050,54.230,160.221
C07962=1014.175,216.566,367.225,168.055,54.220,160.220
C07963=1014.181,216.814,367.200,168.059,54.210,160.219
C07964=1014.186,217.063,367.175,168.064,54.200,160.218
C07965=1014.192,217.312,367.151,168.069,54.189,160.216
C07966=1014.197,217.561,367.126,168.073,54.179,160.215
C07967=1014.202,217.809,367.102,168.078,54.169,160.214
C07968=1014.207,218.057,367.076,168.082,54.159,160.213
C07969=1014.212,218.306,367.052,168.087,54.149,160.212
C07970=1014.218,218.554,367.027,168.092,54.140,160.211
C07971=1014.223,218.802,367.002,168.096,54.129,160.210
C07972=1014.227,219.050,366.978,168.101,54.119,160.208
C07973=1014.233,219.298,366.953,168.106,54.109,160.207
C07974=1014.238,219.546,366.927,168.111,54.100,160.206
C07975=1014.243,219.795,366.903,168.114,54.090,160.205
C07976=1014.249,220.043,366.878,168.119,54.080,160.204
C07977=1014.253,220.292,366.853,168.124,54.070,160.203
C07978=1014.259,220.540,366.828,168.128,54.060,160.202
C07979=1014.264,220.789,366.803,168.133,54.050,160.201
C07980=1014.270,221.037,366.778,168.138,54.041,160.200
C07981=1014.274,221.286,366.753,168.142,54.030,160.198
C07982=1014.279,221.536,366.728,168.147,54.020,160.197
C07983=1014.285,221.784,366.703,168.152,54.011,160.196
C07984=1014.290,222.033,366.678,168.156,54.001,160.195
C07985=1014.296,222.281,366.653,168.161,53.992,160.194
C07986=1014.300,222.530,366.628,168.165,53.982,160.193
C07987=1014.306,222.778,366.603,168.170,53.972,160.192
C07988=1014.311,223.028,366.578,168.175,53.962,160.191
C07989=1014.317,223.276,366.553,168.180,53.953,160.190
C07990=1014.322,223.525,366.527,168.184,53.942,160.188
C07991=1014.328,223.773,366.503,168.188,53.933,160.187
C07992=1014.332,224.022,366.477,168.193,53.923,160.186
C07993=1014.338,224.271,366.452,168.198,53.913,160.185
C07994=1014.343,224.519,366.427,168.203,53.903,160.184
C07995=1014.349,224.769,366.402,168.207,53.894,160.183
C07996=1014.354,225.017,366.377,168.212,53.884,160.182
C07997=1014.359,225.266,366.351,168.216,53.875,160.180
C07998=1014.365,225.514,366.326,168.221,53.865,160.179
C07999=1014.370,225.763,366.301,168.226,53.856,160.179
C08000=1014.376,226.011,366.276,168.231,53.846,160.178
C08001=1014.380,226.260,366.251,168.235,53.837,160.176
C08002=1014.386,226.509,366.225,168.240,53.827,160.175
C08003=1014.391,226.757,366.200,168.245,53.817,160.174
C08004=1014.397,227.006,366.174,168.250,53.808,160.173
C08005=1014.402,227.254,366.148,168.254,53.799,160.172
C08006=1014.407,227.504,366.123,168.259,53.789,160.171
C08007=1014.412,227.752,366.098,168.264,53.779,160.170
C08008=1014.418,228.001,366.072,168.268,53.770,160.169
C08009=1014.423,228.249,366.047,168.273,53.761,160.168
C08010=1014.428,228.498,366.021,168.278,53.751,160.167
C08011=1014.433,228.747,365.995,168.282,53.742,160.166
C08012=1014.439,228.995,365.969,168.287,53.733,160.165
C08013=1014.444,229.243,365.944,168.292,53.723,160.164
C08014=1014.449,229.493,365.919,168.296,53.714,160.163
C08015=1014.454,229.741,365.893,168.301,53.705,160.162
C08016=1014.460,229.990,365.867,168.306,53.695,160.161
C08017=1014.465,230.238,365.841,168.310,53.687,160.160
C08018=1014.470,230.487,365.815,168.315,53.677,160.159
C08019=1014.476,230.736,365.789,168.320,53.667,160.158
C08020=1014.481,230.984,365.764,168.324,53.659,160.157
C08021=1014.486,231.233,365.738,168.329,53.649,160.156
C08022=1014.491,231.481,365.712,168.334,53.640,160.155
C08023=1014.497,231.730,365.686,168.339,53.631,160.154
C08024=1014.502,231.978,365.661,168.343,53.622,160.153
C08025=1014.508,232.227,365.635,168.348,53.613,160.152
C08026=1014.513,232.476,365.610,168.353,53.603,160.151
C08027=1014.518,232.725,365.584,168.358,53.595,160.150
C08028=1014.524,232.973,365.557,168.362,53.585,160.149
C08029=1014.528,233.218,365.532,168.367,53.577,160.148
C08030=1014.534,233.461,365.507,168.372,53.568,160.147
C08031=1014.539,233.705,365.481,168.377,53.559,160.146
C08032=1014.545,233.948,365.456,168.380,53.550,160.145
C08033=1014.550,234.194,365.430,168.386,53.541,160.144
C08034=1014.555,234.437,365.405,168.390,53.532,160.143
C08035=1014.561,234.681,365.379,168.396,53.523,160.142
C08036=1014.566,234.925,365.354,168.400,53.514,160.141
C08037=1014.571,235.174,365.328,168.404,53.505,160.140
C08038=1014.576,235.422,365.302,168.409,53.496,160.139
C08039=1014.582,235.671,365.276,168.414,53.488,160.138
C08040=1014.588,235.919,365.250,168.419,53.478,160.137
C08041=1014.592,236.167,365.224,168.423,53.469,160.136
C08042=1014.598,236.416,365.198,168.428,53.460,160.136
C08043=1014.604,236.665,365.172,168.433,53.452,160.135
C08044=1014.609,236.914,365.146,168.438,53.442,160.134
C08045=1014.614,237.161,365.119,168.442,53.434,160.133
C08046=1014.620,237.410,365.093,168.447,53.425,160.132
C08047=1014.625,237.659,365.067,168.452,53.416,160.131
C08048=1014.631,237.908,365.041,168.457,53.407,160.130
C08049=1014.636,238.156,365.015,168.462,53.399,160.129
C08050=1014.642,238.404,364.989,168.467,53.390,160.128
C08051=1014.646,238.654,364.962,168.471,53.380,160.127
C08052=1014.652,238.902,364.935,168.476,53.371,160.126
C08053=1014.657,239.150,364.910,168.481,53.363,160.125
C08054=1014.663,239.399,364.883,168.485,53.354,160.124
C08055=1014.668,239.647,364.856,168.491,53.346,160.124
C08056=1014.673,239.896,364.830,168.496,53.337,160.123
C08057=1014.679,240.145,364.803,168.500,53.329,160.122
C08058=1014.684,240.393,364.776,168.505,53.320,160.121
C08059=1014.689,240.642,364.751,168.510,53.311,160.120
C08060=1014.695,240.890,364.724,168.515,53.303,160.119
C08061=1014.701,241.138,364.697,168.520,53.294,160.118
C08062=1014.705,241.388,364.671,168.524,53.285,160.117
C08063=1014.711,241.636,364.644,168.529,53.276,160.116
C08064=1014.717,241.884,364.617,168.534,53.268,160.115
C08065=1014.721,242.132,364.591,168.539,53.260,160.115
C08066=1014.727,242.381,364.565,168.544,53.251,160.114
C08067=1014.733,242.630,364.538,168.549,53.243,160.113
C08068=1014.738,242.878,364.511,168.553,53.234,160.112
C08069=1014.743,243.127,364.484,168.558,53.226,160.111
C08070=1014.748,243.375,364.457,168.563,53.217,160.110
C08071=1014.754,243.624,364.430,168.568,53.209,160.110
C08072=1014.759,243.872,364.403,168.573,53.201,160.109
C08073=1014.764,244.120,364.376,168.577,53.192,160.108
C08074=1014.769,244.369,364.349,168.583,53.184,160.107
C08075=1014.774,244.617,364.322,168.587,53.176,160.106
C08076=1014.780,244.866,364.296,168.592,53.167,160.105
C08077=1014.785,245.114,364.268,168.597,53.159,160.105
C08078=1014.791,245.363,364.242,168.601,53.151,160.104
C08079=1014.796,245.611,364.214,168.607,53.143,160.103
C08080=1014.801,245.860,364.187,168.612,53.134,160.102
C08081=1014.807,246.109,364.161,168.617,53.126,160.101
C08082=1014.812,246.357,364.133,168.621,53.118,160.100
C08083=1014.818,246.606,364.107,168.626,53.110,160.100
C08084=1014.823,246.854,364.079,168.631,53.101,160.099
C08085=1014.828,247.103,364.052,168.636,53.093,160.098
C08086=1014.834,247.351,364.026,168.641,53.085,160.097
C08087=1014.839,247.599,363.998,168.646,53.077,160.097
C08088=1014.845,247.848,363.971,168.650,53.068,160.096
C08089=1014.850,248.089,363.945,168.655,53.060,160.095
C08090=1014.855,248.329,363.918,168.660,53.053,160.094
C08091=1014.860,248.570,363.892,168.665,53.045,160.093
C08092=1014.866,248.810,363.866,168.670,53.037,160.093
C08093=1014.870,249.051,363.839,168.675,53.029,160.092
C08094=1014.876,249.291,363.813,168.680,53.021,160.091
C08095=1014.881,249.532,363.787,168.684,53.013,160.090
C08096=1014.886,249.772,363.760,168.689,53.005,160.090
C08097=1014.891,250.021,363.733,168.694,52.997,160.089
C08098=1014.897,250.269,363.706,168.699,52.989,160.088
C08099=1014.903,250.517,363.678,168.703,52.981,160.087
C08100=1014.908,250.766,363.652,168.708,52.973,160.086
C08101=1014.914,251.015,363.624,168.713,52.965,160.086
C08102=1014.919,251.264,363.597,168.719,52.957,160.085
C08103=1014.925,251.511,363.570,168.723,52.949,160.084
C08104=1014.930,251.760,363.542,168.728,52.941,160.083
C08105=1014.936,252.008,363.516,168.733,52.933,160.083
C08106=1014.941,252.256,363.488,168.738,52.925,160.082
C08107=1014.947,252.506,363.460,168.743,52.917,160.081
C08108=1014.953,252.753,363.433,168.748,52.909,160.080
C08109=1014.958,253.002,363.406,168.754,52.901,160.080
C08110=1014.964,253.251,363.379,168.759,52.893,160.079
C08111=1014.969,253.499,363.351,168.763,52.885,160.078
C08112=1014.975,253.748,363.323,168.768,52.878,160.078
C08113=1014.981,253.996,363.296,168.773,52.870,160.077
C08114=1014.986,254.244,363.269,168.778,52.861,160.076
C08115=1014.992,254.492,363.241,168.783,52.854,160.075
C08116=1014.998,254.741,363.214,168.788,52.846,160.074
C08117=1015.003,254.990,363.186,168.793,52.838,160.074
C08118=1015.009,255.238,363.159,168.799,52.830,160.073
C08119=1015.014,255.486,363.131,168.804,52.822,160.072
C08120=1015.020,255.735,363.104,168.809,52.814,160.072
C08121=1015.026,255.983,363.076,168.813,52.806,160.071
C08122=1015.031,256.232,363.049,168.818,52.799,160.070
C08123=1015.037,256.480,363.021,168.823,52.791,160.070
C08124=1015.043,256.729,362.994,168.828,52.783,160.069
C08125=1015.048,256.977,362.966,168.833,52.775,160.068
C08126=1015.055,257.225,362.938,168.838,52.768,160.067
C08127=1015.060,257.474,362.911,168.843,52.760,160.067
C08128=1015.066,257.722,362.884,168.849,52.752,160.066
C08129=1015.071,257.971,362.856,168.854,52.744,160.065
C08130=1015.077,258.219,362.828,168.859,52.736,160.065
C08131=1015.083,258.467,362.801,168.864,52.729,160.064
C08132=1015.088,258.716,362.773,168.869,52.721,160.063
C08133=1015.094,258.964,362.746,168.874,52.714,160.063
C08134=1015.100,259.212,362.718,168.879,52.706,160.062
C08135=1015.106,259.460,362.690,168.884,52.698,160.061
C08136=1015.112,259.709,362.662,168.889,52.690,160.060
C08137=1015.117,259.957,362.634,168.895,52.683,160.060
C08138=1015.123,260.205,362.606,168.900,52.676,160.059
C08139=1015.128,260.453,362.578,168.905,52.668,160.059
C08140=1015.134,260.702,362.549,168.910,52.661,160.058
C08141=1015.139,260.951,362.521,168.915,52.653,160.057
C08142=1015.144,261.199,362.493,168.920,52.646,160.057
C08143=1015.150,261.447,362.465,168.925,52.638,160.056
C08144=1015.156,261.695,362.437,168.930,52.631,160.055
C08145=1015.162,261.944,362.408,168.935,52.624,160.055
C08146=1015.167,262.192,362.380,168.940,52.617,160.054
C08147=1015.173,262.441,362.352,168.945,52.609,160.053
C08148=1015.178,262.689,362.324,168.951,52.602,160.053
C08149=1015.184,262.929,362.297,168.956,52.594,160.052
C08150=1015.190,263.168,362.270,168.960,52.587,160.052
C08151=1015.195,263.408,362.243,168.965,52.580,160.051
C08152=1015.200,263.647,362.216,168.971,52.573,160.051
C08153=1015.206,263.887,362.188,168.975,52.566,160.050
C08154=1015.211,264.127,362.161,168.980,52.559,160.049
C08155=1015.217,264.366,362.133,168.986,52.552,160.049
C08156=1015.223,264.606,362.106,168.990,52.545,160.048
C08157=1015.227,264.854,362.078,168.996,52.538,160.048
C08158=1015.233,265.103,362.049,169.001,52.530,160.047
C08159=1015.239,265.350,362.021,169.006,52.523,160.046
C08160=1015.245,265.599,361.992,169.011,52.516,160.046
C08161=1015.250,265.847,361.964,169.016,52.509,160.045
C08162=1015.257,266.095,361.935,169.021,52.502,160.045
C08163=1015.261,266.344,361.907,169.026,52.495,160.044
C08164=1015.267,266.592,361.878,169.032,52.488,160.044
C08165=1015.273,266.840,361.849,169.037,52.480,160.043
C08166=1015.279,267.089,361.821,169.042,52.473,160.042
C08167=1015.285,267.337,361.792,169.048,52.466,160.042
C08168=1015.290,267.585,361.764,169.052,52.460,160.041
C08169=1015.295,267.834,361.735,169.057,52.452,160.041
C08170=1015.302,268.082,361.706,169.063,52.445,160.040
C08171=1015.307,268.330,361.678,169.068,52.438,160.040
C08172=1015.313,268.578,361.649,169.073,52.431,160.039
C08173=1015.319,268.827,361.620,169.079,52.424,160.039
C08174=1015.324,269.075,361.592,169.083,52.417,160.038
C08175=1015.330,269.323,361.563,169.089,52.410,160.037
C08176=1015.336,269.572,361.534,169.094,52.403,160.037
C08177=1015.341,269.819,361.505,169.099,52.396,160.036
C08178=1015.346,270.068,361.476,169.105,52.389,160.036
C08179=1015.353,270.316,361.447,169.109,52.382,160.035
C08180=1015.358,270.564,361.418,169.115,52.375,160.035
C08181=1015.364,270.813,361.390,169.120,52.368,160.034
C08182=1015.370,271.061,361.361,169.126,52.361,160.034
C08183=1015.375,271.308,361.332,169.131,52.354,160.033
C08184=1015.381,271.558,361.303,169.136,52.348,160.033
C08185=1015.387,271.806,361.274,169.142,52.341,160.032
C08186=1015.392,272.054,361.244,169.147,52.334,160.032
C08187=1015.398,272.302,361.216,169.152,52.327,160.031
C08188=1015.404,272.550,361.187,169.157,52.321,160.031
C08189=1015.410,272.799,361.158,169.162,52.314,160.030
C08190=1015.416,273.047,361.129,169.168,52.307,160.030
C08191=1015.421,273.295,361.099,169.174,52.300,160.029
C08192=1015.427,273.543,361.070,169.178,52.294,160.029
C08193=1015.432,273.791,361.041,169.184,52.287,160.028
C08194=1015.439,274.039,361.012,169.189,52.280,160.028
C08195=1015.444,274.288,360.982,169.195,52.273,160.028
C08196=1015.450,274.536,360.954,169.199,52.267,160.027
C08197=1015.455,274.784,360.924,169.205,52.260,160.026
C08198=1015.461,275.032,360.895,169.211,52.253,160.026
C08199=1015.467,275.281,360.866,169.215,52.247,160.026
C08200=1015.473,275.529,360.837,169.221,52.240,160.025
C08201=1015.479,275.777,360.807,169.227,52.233,160.025
C08202=1015.485,276.026,360.778,169.232,52.226,160.024
C08203=1015.490,276.274,360.748,169.237,52.221,160.024
C08204=1015.496,276.521,360.719,169.242,52.214,160.023
C08205=1015.502,276.769,360.689,169.248,52.207,160.023
C08206=1015.507,277.018,360.660,169.253,52.201,160.022
C08207=1015.514,277.266,360.631,169.259,52.194,160.022
C08208=1015.519,277.514,360.601,169.264,52.187,160.022
C08209=1015.524,277.756,360.572,169.269,52.181,160.021
C08210=1015.530,277.997,360.543,169.275,52.175,160.021
C08211=1015.536,278.239,360.514,169.279,52.168,160.020
C08212=1015.541,278.481,360.485,169.284,52.163,160.020
C08213=1015.547,278.723,360.457,169.290,52.156,160.020
C08214=1015.553,278.965,360.428,169.295,52.150,160.019
C08215=1015.558,279.206,360.399,169.301,52.144,160.019
C08216=1015.565,279.449,360.369,169.305,52.137,160.018
C08217=1015.570,279.697,360.340,169.311,52.131,160.018
C08218=1015.576,279.945,360.310,169.317,52.125,160.018
C08219=1015.582,280.193,360.280,169.322,52.118,160.017
C08220=1015.588,280.441,360.251,169.328,52.112,160.017
C08221=1015.593,280.690,360.221,169.334,52.106,160.017
C08222=1015.599,280.938,360.191,169.338,52.100,160.016
C08223=1015.605,281.186,360.162,169.344,52.093,160.016
C08224=1015.611,281.434,360.131,169.350,52.086,160.015
C08225=1015.617,281.682,360.102,169.355,52.080,160.015
C08226=1015.622,281.931,360.072,169.361,52.074,160.015
C08227=1015.629,282.178,360.042,169.365,52.068,160.014
C08228=1015.634,282.426,360.013,169.371,52.061,160.014
C08229=1015.640,282.674,359.982,169.377,52.055,160.013
C08230=1015.646,282.922,359.953,169.382,52.049,160.013
C08231=1015.652,283.170,359.923,169.388,52.043,160.013
C08232=1015.658,283.419,359.893,169.394,52.037,160.012
C08233=1015.664,283.667,359.862,169.399,52.031,160.012
C08234=1015.670,283.915,359.833,169.405,52.024,160.012
C08235=1015.676,284.163,359.803,169.410,52.017,160.011
C08236=1015.682,284.411,359.773,169.415,52.011,160.011
C08237=1015.688,284.659,359.742,169.421,52.005,160.011
C08238=1015.693,284.907,359.713,169.426,51.999,160.010
C08239=1015.699,285.155,359.682,169.432,51.994,160.010
C08240=1015.705,285.404,359.652,169.438,51.987,160.010
C08241=1015.711,285.651,359.621,169.443,51.982,160.009
C08242=1015.717,285.900,359.592,169.449,51.975,160.009
C08243=1015.723,286.148,359.561,169.454,51.969,160.009
C08244=1015.728,286.395,359.531,169.460,51.963,160.008
C08245=1015.736,286.644,359.501,169.465,51.957,160.008
C08246=1015.741,286.892,359.471,169.471,51.951,160.008
C08247=1015.747,287.139,359.440,169.476,51.945,160.007
C08248=1015.753,287.387,359.410,169.482,51.939,160.007
C08249=1015.759,287.635,359.379,169.488,51.933,160.007
C08250=1015.764,287.884,359.348,169.493,51.927,160.006
C08251=1015.770,288.132,359.319,169.499,51.921,160.006
C08252=1015.776,288.380,359.288,169.504,51.916,160.006
C08253=1015.782,288.629,359.257,169.510,51.909,160.006
C08254=1015.788,288.876,359.227,169.516,51.903,160.005
C08255=1015.794,289.124,359.197,169.521,51.898,160.005
C08256=1015.800,289.373,359.166,169.527,51.892,160.005
C08257=1015.806,289.620,359.135,169.532,51.886,160.005
C08258=1015.812,289.868,359.105,169.538,51.880,160.004
C08259=1015.818,290.116,359.074,169.543,51.874,160.004
C08260=1015.824,290.364,359.044,169.549,51.868,160.004
C08261=1015.830,290.612,359.013,169.555,51.863,160.004
C08262=1015.837,290.860,358.982,169.560,51.857,160.003
C08263=1015.842,291.108,358.952,169.567,51.851,160.003
C08264=1015.849,291.356,358.921,169.572,51.845,160.003
C08265=1015.854,291.604,358.890,169.578,51.840,160.003
C08266=1015.860,291.852,358.859,169.583,51.834,160.002
C08267=1015.866,292.100,358.829,169.589,51.828,160.002
C08268=1015.873,292.348,358.798,169.594,51.822,160.002
C08269=1015.878,292.596,358.767,169.601,51.817,160.002
C08270=1015.884,292.844,358.736,169.606,51.811,160.001
C08271=1015.890,293.092,358.705,169.612,51.805,160.001
C08272=1015.895,293.340,358.674,169.617,51.800,160.001
C08273=1015.902,293.588,358.643,169.624,51.794,160.001
C08274=1015.907,293.836,358.612,169.629,51.789,160.001
C08275=1015.913,294.083,358.580,169.635,51.783,160.000
C08276=1015.919,294.331,358.548,169.640,51.778,160.000
C08277=1015.925,294.579,358.518,169.646,51.773,160.000
C08278=1015.931,294.827,358.486,169.652,51.766,160.000
C08279=1015.937,295.075,358.456,169.657,51.761,160.000
C08280=1015.943,295.323,358.424,169.663,51.756,160.000
C08281=1015.949,295.571,358.393,169.669,51.750,159.999
C08282=1015.955,295.819,358.361,169.675,51.745,159.999
C08283=1015.961,296.067,358.330,169.680,51.740,159.999
C08284=1015.967,296.315,358.298,169.687,51.734,159.999
C08285=1015.973,296.563,358.268,169.692,51.728,159.999
C08286=1015.979,296.811,358.236,169.698,51.723,159.998
C08287=1015.984,297.058,358.204,169.703,51.717,159.998
C08288=1015.991,297.306,358.173,169.709,51.712,159.998
C08289=1015.996,297.555,358.141,169.715,51.707,159.998
C08290=1016.003,297.802,358.110,169.720,51.701,159.998
C08291=1016.008,298.051,358.078,169.727,51.696,159.998
C08292=1016.015,298.298,358.047,169.732,51.691,159.998
C08293=1016.021,298.546,358.015,169.739,51.685,159.997
C08294=1016.026,298.794,357.985,169.744,51.680,159.997
C08295=1016.032,299.042,357.953,169.750,51.674,159.997
C08296=1016.039,299.290,357.921,169.756,51.669,159.997
C08297=1016.045,299.537,357.890,169.762,51.664,159.997
C08298=1016.051,299.785,357.858,169.767,51.658,159.997
C08299=1016.057,300.034,357.826,169.774,51.653,159.997
C08300=1016.063,300.281,357.795,169.780,51.648,159.997
C08301=1016.069,300.529,357.763,169.785,51.643,159.996
C08302=1016.075,300.777,357.731,169.791,51.638,159.996
C08303=1016.082,301.025,357.700,169.797,51.632,159.996
C08304=1016.087,301.273,357.668,169.803,51.627,159.996
C08305=1016.094,301.520,357.637,169.809,51.622,159.996
C08306=1016.100,301.769,357.605,169.815,51.617,159.996
C08307=1016.107,302.017,357.573,169.821,51.612,159.996
C08308=1016.112,302.264,357.542,169.827,51.606,159.996
C08309=1016.119,302.512,357.510,169.832,51.601,159.995
C08310=1016.125,302.760,357.478,169.839,51.596,159.996
C08311=1016.132,303.008,357.447,169.844,51.591,159.995
C08312=1016.137,303.256,357.415,169.851,51.585,159.995
C08313=1016.143,303.503,357.382,169.857,51.581,159.995
C08314=1016.150,303.751,357.351,169.863,51.575,159.995
C08315=1016.156,303.999,357.319,169.868,51.570,159.995
C08316=1016.163,304.247,357.287,169.875,51.565,159.995
C08317=1016.169,304.495,357.255,169.880,51.560,159.995
C08318=1016.176,304.743,357.223,169.887,51.554,159.995
C08319=1016.181,304.990,357.192,169.893,51.550,159.995
C08320=1016.188,305.238,357.160,169.899,51.544,159.995
C08321=1016.194,305.486,357.128,169.905,51.540,159.995
C08322=1016.201,305.734,357.096,169.911,51.534,159.995
C08323=1016.207,305.982,357.064,169.916,51.529,159.994
C08324=1016.213,306.230,357.032,169.923,51.524,159.995
C08325=1016.220,306.477,357.000,169.929,51.519,159.994
C08326=1016.226,306.726,356.968,169.935,51.514,159.995
C08327=1016.233,306.973,356.936,169.941,51.509,159.994
C08328=1016.239,307.221,356.904,169.948,51.504,159.994
C08329=1016.246,307.487,356.869,169.954,51.499,159.994
C08330=1016.253,307.753,356.835,169.960,51.493,159.994
C08331=1016.260,308.019,356.800,169.967,51.488,159.994
C08332=1016.267,308.284,356.766,169.974,51.483,159.994
C08333=1016.274,308.532,356.734,169.979,51.478,159.994
C08334=1016.280,308.780,356.702,169.986,51.473,159.994
C08335=1016.287,309.028,356.670,169.991,51.468,159.994
C08336=1016.293,309.275,356.637,169.998,51.463,159.994
C08337=1016.299,309.523,356.605,170.004,51.458,159.994
C08338=1016.305,309.771,356.573,170.010,51.453,159.994
C08339=1016.312,310.019,356.540,170.016,51.449,159.994
C08340=1016.318,310.266,356.507,170.022,51.444,159.994
C08341=1016.324,310.514,356.474,170.029,51.439,159.994
C08342=1016.330,310.762,356.441,170.035,51.435,159.994
C08343=1016.336,311.009,356.408,170.041,51.430,159.994
C08344=1016.342,311.257,356.376,170.047,51.426,159.994
C08345=1016.349,311.505,356.343,170.053,51.421,159.994
C08346=1016.355,311.752,356.310,170.060,51.416,159.995
C08347=1016.360,312.000,356.277,170.066,51.412,159.995
C08348=1016.367,312.248,356.244,170.071,51.407,159.995
C08349=1016.373,312.495,356.211,170.078,51.402,159.995
C08350=1016.379,312.743,356.179,170.084,51.398,159.995
C08351=1016.386,312.991,356.145,170.091,51.393,159.995
C08352=1016.392,313.239,356.112,170.096,51.388,159.995
C08353=1016.398,313.486,356.079,170.103,51.385,159.995
C08354=1016.405,313.734,356.046,170.110,51.380,159.995
C08355=1016.411,313.981,356.013,170.115,51.375,159.995
C08356=1016.418,314.229,355.980,170.122,51.370,159.995
C08357=1016.423,314.477,355.947,170.128,51.366,159.995
C08358=1016.430,314.725,355.914,170.135,51.361,159.995
C08359=1016.436,314.972,355.881,170.141,51.357,159.996
C08360=1016.443,315.220,355.848,170.147,51.353,159.996
C08361=1016.449,315.468,355.815,170.153,51.348,159.996
C08362=1016.455,315.716,355.781,170.159,51.343,159.996
C08363=1016.462,315.963,355.748,170.166,51.339,159.996
C08364=1016.468,316.211,355.715,170.172,51.335,159.996
C08365=1016.475,316.459,355.682,170.178,51.330,159.996
C08366=1016.481,316.706,355.649,170.185,51.326,159.996
C08367=1016.488,316.954,355.615,170.191,51.322,159.996
C08368=1016.494,317.202,355.582,170.198,51.317,159.997
C08369=1016.500,317.449,355.549,170.204,51.313,159.997
C08370=1016.507,317.697,355.516,170.211,51.308,159.997
C08371=1016.513,317.944,355.481,170.217,51.304,159.997
C08372=1016.519,318.192,355.449,170.224,51.299,159.997
C08373=1016.527,318.440,355.415,170.230,51.295,159.997
C08374=1016.533,318.687,355.382,170.236,51.291,159.997
C08375=1016.540,318.935,355.348,170.243,51.286,159.998
C08376=1016.546,319.183,355.315,170.249,51.282,159.998
C08377=1016.553,319.430,355.281,170.256,51.278,159.998
C08378=1016.559,319.678,355.248,170.262,51.274,159.998
C08379=1016.566,319.926,355.215,170.269,51.269,159.998
C08380=1016.572,320.174,355.181,170.275,51.265,159.998
C08381=1016.579,320.421,355.147,170.282,51.260,159.999
C08382=1016.586,320.668,355.114,170.288,51.256,159.999
C08383=1016.593,320.917,355.081,170.295,51.252,159.999
C08384=1016.599,321.163,355.047,170.301,51.248,159.999
C08385=1016.606,321.411,355.013,170.308,51.244,159.999
C08386=1016.612,321.659,354.980,170.314,51.239,159.999
C08387=1016.619,321.907,354.946,170.321,51.235,160.000
C08388=1016.626,322.154,354.913,170.327,51.231,160.000
C08389=1016.634,322.426,354.876,170.334,51.226,160.000
C08390=1016.640,322.696,354.839,170.341,51.222,160.000
C08391=1016.648,322.969,354.802,170.349,51.217,160.000
C08392=1016.656,323.239,354.765,170.356,51.213,160.001
C08393=1016.662,323.487,354.732,170.362,51.209,160.001
C08394=1016.669,323.735,354.698,170.369,51.204,160.001
C08395=1016.676,323.982,354.664,170.375,51.200,160.001
C08396=1016.682,324.230,354.630,170.383,51.196,160.002
C08397=1016.689,324.477,354.596,170.389,51.192,160.002
C08398=1016.697,324.725,354.563,170.396,51.188,160.002
C08399=1016.703,324.972,354.529,170.402,51.184,160.002
C08400=1016.710,325.220,354.495,170.409,51.179,160.002
C08401=1016.717,325.468,354.461,170.415,51.176,160.003
C08402=1016.724,325.715,354.427,170.422,51.171,160.003
C08403=1016.731,325.962,354.394,170.430,51.167,160.003
C08404=1016.737,326.210,354.359,170.436,51.164,160.004
C08405=1016.744,326.458,354.325,170.442,51.160,160.004
C08406=1016.751,326.705,354.290,170.449,51.156,160.004
C08407=1016.757,326.953,354.256,170.456,51.152,160.004
C08408=1016.764,327.200,354.222,170.463,51.148,160.005
C08409=1016.771,327.448,354.187,170.469,51.144,160.005
C08410=1016.777,327.696,354.153,170.477,51.140,160.005
C08411=1016.785,327.943,354.119,170.483,51.136,160.005
C08412=1016.791,328.191,354.084,170.490,51.132,160.006
C08413=1016.797,328.438,354.050,170.496,51.128,160.006
C08414=1016.804,328.686,354.015,170.504,51.125,160.007
C08415=1016.811,328.933,353.981,170.510,51.121,160.007
C08416=1016.818,329.181,353.946,170.517,51.117,160.007
C08417=1016.824,329.428,353.911,170.524,51.114,160.007
C08418=1016.832,329.676,353.877,170.531,51.110,160.008
C08419=1016.838,329.923,353.842,170.537,51.106,160.008
C08420=1016.845,330.171,353.808,170.545,51.102,160.009
C08421=1016.852,330.418,353.773,170.551,51.098,160.009
C08422=1016.859,330.666,353.738,170.558,51.094,160.009
C08423=1016.866,330.914,353.704,170.565,51.091,160.009
C08424=1016.873,331.161,353.669,170.572,51.087,160.010
C08425=1016.880,331.409,353.635,170.579,51.084,160.010
C08426=1016.886,331.656,353.600,170.586,51.080,160.010
C08427=1016.894,331.903,353.565,170.592,51.076,160.011
C08428=1016.900,332.151,353.531,170.600,51.072,160.011
C08429=1016.907,332.399,353.496,170.606,51.069,160.011
C08430=1016.914,332.646,353.460,170.614,51.065,160.012
C08431=1016.921,332.893,353.425,170.620,51.062,160.012
C08432=1016.927,333.141,353.390,170.627,51.058,160.013
C08433=1016.934,333.388,353.355,170.634,51.055,160.013
C08434=1016.941,333.635,353.320,170.642,51.051,160.014
C08435=1016.948,333.882,353.285,170.648,51.047,160.014
C08436=1016.955,334.130,353.250,170.655,51.044,160.014
C08437=1016.962,334.377,353.215,170.662,51.041,160.015
C08438=1016.969,334.625,353.180,170.669,51.036,160.015
C08439=1016.976,334.873,353.144,170.676,51.033,160.015
C08440=1016.983,335.120,353.109,170.683,51.030,160.016
C08441=1016.990,335.367,353.074,170.690,51.027,160.016
C08442=1016.996,335.615,353.039,170.697,51.022,160.017
C08443=1017.003,335.862,353.004,170.704,51.019,160.017
C08444=1017.010,336.110,352.968,170.711,51.016,160.018
C08445=1017.017,336.357,352.933,170.718,51.013,160.018
C08446=1017.024,336.605,352.898,170.726,51.009,160.019
C08447=1017.031,336.852,352.862,170.732,51.006,160.019
C08448=1017.038,337.100,352.827,170.740,51.002,160.019
C08449=1017.046,337.366,352.789,170.747,50.998,160.020
C08450=1017.053,337.634,352.751,170.755,50.995,160.020
C08451=1017.061,337.900,352.713,170.762,50.991,160.021
C08452=1017.069,338.167,352.674,170.771,50.987,160.021
C08453=1017.076,338.414,352.639,170.778,50.984,160.022
C08454=1017.083,338.662,352.604,170.785,50.981,160.022
C08455=1017.090,338.909,352.568,170.792,50.978,160.023
C08456=1017.096,339.157,352.532,170.799,50.974,160.023
C08457=1017.104,339.404,352.496,170.806,50.971,160.024
C08458=1017.111,339.652,352.461,170.814,50.968,160.024
C08459=1017.118,339.898,352.425,170.821,50.965,160.025
C08460=1017.125,340.146,352.389,170.828,50.961,160.025
C08461=1017.132,340.393,352.353,170.836,50.958,160.026
C08462=1017.139,340.641,352.317,170.842,50.955,160.026
C08463=1017.146,340.888,352.281,170.850,50.952,160.027
C08464=1017.153,341.135,352.246,170.857,50.949,160.027
C08465=1017.161,341.382,352.209,170.865,50.945,160.028
C08466=1017.167,341.630,352.174,170.872,50.943,160.028
C08467=1017.175,341.878,352.137,170.879,50.939,160.029
C08468=1017.182,342.124,352.102,170.887,50.936,160.029
C08469=1017.189,342.372,352.065,170.894,50.933,160.030
C08470=1017.196,342.619,352.030,170.902,50.930,160.031
C08471=1017.203,342.867,351.993,170.908,50.926,160.031
C08472=1017.210,343.114,351.958,170.916,50.924,160.032
C08473=1017.218,343.361,351.921,170.924,50.920,160.032
C08474=1017.225,343.609,351.885,170.931,50.918,160.033
C08475=1017.232,343.856,351.849,170.938,50.914,160.033
C08476=1017.239,344.103,351.812,170.945,50.912,160.034
C08477=1017.246,344.350,351.776,170.953,50.908,160.034
C08478=1017.254,344.597,351.740,170.961,50.905,160.035
C08479=1017.261,344.845,351.704,170.968,50.903,160.036
C08480=1017.268,345.092,351.668,170.976,50.899,160.036
C08481=1017.275,345.339,351.631,170.984,50.896,160.037
C08482=1017.283,345.587,351.595,170.990,50.893,160.037
C08483=1017.290,345.834,351.559,170.998,50.890,160.038
C08484=1017.297,346.081,351.522,171.005,50.888,160.039
C08485=1017.305,346.328,351.485,171.013,50.884,160.039
C08486=1017.313,346.576,351.449,171.021,50.881,160.040
C08487=1017.319,346.823,351.412,171.028,50.879,160.041
C08488=1017.327,347.070,351.376,171.036,50.876,160.041
C08489=1017.334,347.317,351.339,171.043,50.873,160.042
C08490=1017.341,347.565,351.303,171.050,50.870,160.042
C08491=1017.348,347.812,351.266,171.058,50.867,160.043
C08492=1017.356,348.059,351.229,171.066,50.864,160.044
C08493=1017.363,348.306,351.192,171.073,50.862,160.045
C08494=1017.371,348.553,351.155,171.081,50.859,160.045
C08495=1017.378,348.801,351.119,171.090,50.856,160.046
C08496=1017.385,349.047,351.082,171.097,50.854,160.047
C08497=1017.392,349.295,351.045,171.105,50.851,160.047
C08498=1017.400,349.542,351.008,171.113,50.848,160.048
C08499=1017.407,349.789,350.971,171.120,50.845,160.049
C08500=1017.415,350.036,350.935,171.128,50.842,160.049
C08501=1017.422,350.283,350.897,171.136,50.840,160.050
C08502=1017.429,350.531,350.860,171.144,50.837,160.051
C08503=1017.437,350.778,350.823,171.151,50.834,160.051
C08504=1017.444,351.025,350.786,171.159,50.831,160.052
C08505=1017.452,351.272,350.749,171.167,50.829,160.053
C08506=1017.459,351.520,350.712,171.174,50.827,160.054
C08507=1017.467,351.766,350.675,171.182,50.824,160.054
C08508=1017.474,352.014,350.638,171.190,50.821,160.055
C08509=1017.482,352.278,350.598,171.198,50.818,160.056
C08510=1017.490,352.541,350.559,171.206,50.816,160.057
C08511=1017.499,352.806,350.519,171.215,50.813,160.057
C08512=1017.506,353.070,350.479,171.223,50.810,160.058
C08513=1017.514,353.318,350.442,171.231,50.807,160.059
C08514=1017.521,353.565,350.404,171.240,50.805,160.060
C08515=1017.529,353.812,350.367,171.247,50.802,160.060
C08516=1017.537,354.059,350.330,171.255,50.800,160.061
C08517=1017.544,354.305,350.291,171.263,50.797,160.062
C08518=1017.551,354.553,350.254,171.272,50.795,160.063
C08519=1017.559,354.799,350.217,171.279,50.792,160.064
C08520=1017.567,355.047,350.179,171.287,50.790,160.064
C08521=1017.575,355.294,350.141,171.295,50.787,160.065
C08522=1017.582,355.542,350.104,171.303,50.785,160.066
C08523=1017.590,355.788,350.066,171.311,50.782,160.067
C08524=1017.597,356.035,350.029,171.319,50.780,160.068
C08525=1017.605,356.282,349.991,171.327,50.777,160.068
C08526=1017.613,356.529,349.953,171.335,50.775,160.069
C08527=1017.621,356.776,349.916,171.344,50.773,160.070
C08528=1017.628,357.023,349.878,171.352,50.770,160.071
C08529=1017.635,357.270,349.840,171.360,50.768,160.072
C08530=1017.643,357.518,349.802,171.367,50.766,160.073
C08531=1017.651,357.764,349.764,171.376,50.764,160.074
C08532=1017.658,358.011,349.726,171.384,50.761,160.074
C08533=1017.667,358.258,349.688,171.392,50.759,160.075
C08534=1017.674,358.505,349.651,171.401,50.756,160.076
C08535=1017.682,358.752,349.612,171.409,50.754,160.077
C08536=1017.690,359.000,349.575,171.417,50.752,160.078
C08537=1017.697,359.246,349.536,171.425,50.750,160.079
C08538=1017.705,359.493,349.498,171.433,50.748,160.080
C08539=1017.713,359.740,349.459,171.442,50.746,160.081
C08540=1017.720,359.987,349.422,171.450,50.743,160.081
C08541=1017.728,360.234,349.383,171.458,50.741,160.082
C08542=1017.736,360.481,349.345,171.467,50.739,160.083
C08543=1017.744,360.728,349.307,171.475,50.737,160.084
C08544=1017.752,360.974,349.268,171.484,50.734,160.085
C08545=1017.760,361.222,349.230,171.491,50.732,160.086
C08546=1017.767,361.468,349.191,171.499,50.730,160.087
C08547=1017.775,361.716,349.152,171.508,50.728,160.088
C08548=1017.782,361.962,349.114,171.517,50.726,160.089
C08549=1017.790,362.209,349.075,171.525,50.724,160.090
C08550=1017.798,362.456,349.037,171.533,50.722,160.091
C08551=1017.806,362.703,348.999,171.542,50.720,160.092
C08552=1017.814,362.950,348.960,171.551,50.718,160.093
C08553=1017.822,363.197,348.922,171.559,50.716,160.094
C08554=1017.830,363.443,348.882,171.567,50.714,160.095
C08555=1017.838,363.690,348.844,171.576,50.711,160.095
C08556=1017.846,363.937,348.805,171.585,50.710,160.097
C08557=1017.854,364.184,348.767,171.593,50.707,160.098
C08558=1017.861,364.431,348.727,171.602,50.706,160.099
C08559=1017.869,364.678,348.689,171.610,50.704,160.100
C08560=1017.877,364.925,348.650,171.619,50.702,160.101
C08561=1017.886,365.172,348.611,171.627,50.700,160.102
C08562=1017.893,365.418,348.573,171.636,50.698,160.102
C08563=1017.902,365.665,348.534,171.645,50.696,160.104
C08564=1017.910,365.912,348.495,171.653,50.694,160.105
C08565=1017.918,366.159,348.456,171.662,50.692,160.106
C08566=1017.926,366.405,348.417,171.670,50.690,160.107
C08567=1017.934,366.652,348.378,171.679,50.688,160.108
C08568=1017.942,366.899,348.339,171.688,50.687,160.109
C08569=1017.952,367.171,348.296,171.697,50.685,160.110
C08570=1017.960,367.442,348.253,171.707,50.683,160.111
C08571=1017.969,367.715,348.210,171.717,50.681,160.112
C08572=1017.978,367.986,348.167,171.727,50.679,160.114
C08573=1017.986,368.233,348.127,171.735,50.676,160.115
C08574=1017.994,368.480,348.087,171.744,50.675,160.116
C08575=1018.002,368.726,348.048,171.753,50.673,160.117
C08576=1018.010,368.973,348.008,171.762,50.672,160.118
C08577=1018.019,369.220,347.969,171.770,50.670,160.119
C08578=1018.026,369.467,347.929,171.779,50.668,160.120
C08579=1018.035,369.713,347.890,171.788,50.667,160.121
C08580=1018.043,369.960,347.850,171.798,50.665,160.122
C08581=1018.051,370.207,347.810,171.807,50.663,160.124
C08582=1018.059,370.453,347.771,171.815,50.661,160.125
C08583=1018.067,370.700,347.731,171.824,50.660,160.126
C08584=1018.076,370.947,347.692,171.833,50.658,160.127
C08585=1018.083,371.194,347.652,171.842,50.657,160.128
C08586=1018.092,371.440,347.612,171.851,50.656,160.129
C08587=1018.100,371.686,347.572,171.861,50.654,160.131
C08588=1018.108,371.933,347.533,171.869,50.652,160.132
C08589=1018.117,372.180,347.493,171.878,50.650,160.133
C08590=1018.125,372.427,347.453,171.887,50.649,160.134
C08591=1018.134,372.673,347.413,171.896,50.648,160.135
C08592=1018.141,372.920,347.373,171.906,50.646,160.137
C08593=1018.150,373.167,347.334,171.915,50.644,160.138
C08594=1018.159,373.413,347.293,171.924,50.643,160.139
C08595=1018.167,373.660,347.253,171.933,50.641,160.140
C08596=1018.176,373.906,347.213,171.943,50.640,160.142
C08597=1018.183,374.153,347.173,171.952,50.638,160.143
C08598=1018.193,374.400,347.133,171.960,50.637,160.144
C08599=1018.201,374.647,347.093,171.971,50.635,160.145
C08600=1018.209,374.893,347.053,171.979,50.634,160.146
C08601=1018.219,375.139,347.013,171.989,50.633,160.148
C08602=1018.226,375.386,346.973,171.998,50.631,160.149
C08603=1018.235,375.632,346.933,172.008,50.630,160.150
C08604=1018.244,375.879,346.892,172.017,50.629,160.151
C08605=1018.252,376.126,346.852,172.027,50.627,160.153
C08606=1018.261,376.373,346.811,172.036,50.626,160.154
C08607=1018.269,376.619,346.771,172.045,50.625,160.155
C08608=1018.277,376.865,346.730,172.055,50.623,160.157
C08609=1018.286,377.112,346.689,172.064,50.622,160.158
C08610=1018.294,377.358,346.649,172.073,50.621,160.159
C08611=1018.303,377.605,346.608,172.083,50.619,160.161
C08612=1018.311,377.852,346.567,172.092,50.618,160.162
C08613=1018.320,378.098,346.526,172.102,50.617,160.163
C08614=1018.328,378.344,346.485,172.112,50.616,160.165
C08615=1018.337,378.591,346.445,172.121,50.615,160.166
C08616=1018.345,378.837,346.404,172.131,50.613,160.167
C08617=1018.354,379.084,346.363,172.140,50.612,160.169
C08618=1018.362,379.330,346.322,172.149,50.611,160.170
C08619=1018.372,379.577,346.281,172.160,50.610,160.172
C08620=1018.380,379.824,346.240,172.169,50.609,160.173
C08621=1018.389,380.069,346.199,172.179,50.608,160.174
C08622=1018.397,380.316,346.158,172.188,50.606,160.176
C08623=1018.407,380.563,346.117,172.198,50.605,160.177
C08624=1018.415,380.809,346.076,172.208,50.605,160.179
C08625=1018.424,381.056,346.035,172.218,50.603,160.180
C08626=1018.432,381.302,345.993,172.227,50.602,160.181
C08627=1018.441,381.549,345.952,172.237,50.601,160.183
C08628=1018.450,381.794,345.912,172.247,50.600,160.184
C08629=1018.460,382.089,345.862,172.259,50.598,160.186
C08630=1018.471,382.383,345.813,172.271,50.597,160.188
C08631=1018.482,382.677,345.763,172.283,50.597,160.189
C08632=1018.492,382.971,345.714,172.294,50.595,160.191
C08633=1018.502,383.218,345.674,172.304,50.594,160.193
C08634=1018.510,383.464,345.632,172.315,50.593,160.194
C08635=1018.519,383.710,345.590,172.324,50.592,160.196
C08636=1018.528,383.957,345.548,172.335,50.591,160.197
C08637=1018.538,384.203,345.507,172.345,50.590,160.199
C08638=1018.547,384.449,345.466,172.354,50.590,160.200
C08639=1018.556,384.695,345.424,172.365,50.588,160.202
C08640=1018.564,384.942,345.383,172.375,50.587,160.203
C08641=1018.573,385.189,345.341,172.385,50.587,160.205
C08642=1018.583,385.434,345.299,172.395,50.586,160.206
C08643=1018.592,385.681,345.257,172.405,50.585,160.208
C08644=1018.601,385.927,345.215,172.415,50.584,160.209
C08645=1018.609,386.174,345.174,172.426,50.584,160.211
C08646=1018.619,386.419,345.131,172.436,50.583,160.213
C08647=1018.628,386.666,345.089,172.447,50.582,160.214
C08648=1018.637,386.912,345.048,172.456,50.581,160.216
C08649=1018.646,387.158,345.005,172.466,50.580,160.217
C08650=1018.655,387.405,344.963,172.477,50.579,160.219
C08651=1018.664,387.651,344.922,172.488,50.578,160.220
C08652=1018.674,387.897,344.879,172.499,50.578,160.222
C08653=1018.682,388.143,344.837,172.508,50.578,160.224
C08654=1018.692,388.389,344.795,172.519,50.577,160.225
C08655=1018.702,388.636,344.752,172.529,50.576,160.227
C08656=1018.710,388.882,344.710,172.540,50.575,160.229
C08657=1018.719,389.128,344.667,172.550,50.575,160.230
C08658=1018.728,389.374,344.625,172.561,50.574,160.232
C08659=1018.738,389.621,344.583,172.571,50.574,160.234
C08660=1018.747,389.867,344.540,172.581,50.573,160.235
C08661=1018.756,390.112,344.498,172.592,50.572,160.237
C08662=1018.765,390.359,344.455,172.603,50.572,160.239
C08663=1018.775,390.605,344.412,172.613,50.571,160.240
C08664=1018.784,390.850,344.370,172.624,50.571,160.242
C08665=1018.794,391.097,344.327,172.635,50.570,160.244
C08666=1018.803,391.343,344.285,172.646,50.570,160.246
C08667=1018.813,391.589,344.242,172.657,50.569,160.247
C08668=1018.821,391.835,344.199,172.667,50.569,160.249
C08669=1018.831,392.082,344.156,172.678,50.568,160.251
C08670=1018.840,392.327,344.113,172.689,50.568,160.253
C08671=1018.850,392.574,344.071,172.700,50.567,160.254
C08672=1018.859,392.820,344.028,172.711,50.567,160.256
C08673=1018.869,393.066,343.984,172.721,50.567,160.258
C08674=1018.877,393.312,343.941,172.732,50.566,160.260
C08675=1018.887,393.558,343.898,172.743,50.566,160.261
C08676=1018.897,393.804,343.855,172.754,50.565,160.263
C08677=1018.906,394.050,343.812,172.765,50.565,160.265
C08678=1018.916,394.296,343.768,172.776,50.565,160.267
C08679=1018.926,394.542,343.725,172.787,50.565,160.269
C08680=1018.935,394.788,343.682,172.799,50.564,160.271
C08681=1018.945,395.034,343.638,172.810,50.564,160.272
C08682=1018.955,395.280,343.595,172.821,50.563,160.274
C08683=1018.963,395.525,343.552,172.832,50.563,160.276
C08684=1018.973,395.772,343.509,172.843,50.563,160.278
C08685=1018.983,396.018,343.465,172.853,50.563,160.280
C08686=1018.993,396.264,343.421,172.865,50.562,160.282
C08687=1019.003,396.510,343.378,172.876,50.562,160.284
C08688=1019.012,396.756,343.334,172.888,50.562,160.286
C08689=1019.025,397.087,343.275,172.903,50.562,160.288
C08690=1019.039,397.419,343.216,172.918,50.562,160.291
C08691=1019.051,397.750,343.157,172.934,50.561,160.293
C08692=1019.065,398.082,343.098,172.949,50.561,160.296
C08693=1019.075,398.328,343.055,172.960,50.561,160.298
C08694=1019.085,398.574,343.010,172.972,50.561,160.300
C08695=1019.094,398.820,342.966,172.983,50.561,160.302
C08696=1019.104,399.066,342.922,172.995,50.560,160.304
C08697=1019.114,399.312,342.878,173.007,50.561,160.306
C08698=1019.124,399.557,342.834,173.018,50.560,160.308
C08699=1019.134,399.803,342.790,173.030,50.560,160.310
C08700=1019.143,400.049,342.745,173.041,50.561,160.312
C08701=1019.153,400.295,342.702,173.053,50.560,160.314
C08702=1019.163,400.541,342.658,173.065,50.560,160.316
C08703=1019.173,400.786,342.613,173.076,50.561,160.318
C08704=1019.184,401.032,342.568,173.088,50.561,160.320
C08705=1019.193,401.278,342.524,173.100,50.561,160.322
C08706=1019.203,401.524,342.479,173.112,50.561,160.324
C08707=1019.212,401.769,342.434,173.123,50.561,160.326
C08708=1019.223,402.015,342.390,173.136,50.561,160.328
C08709=1019.233,402.261,342.345,173.147,50.562,160.331
C08710=1019.243,402.507,342.301,173.159,50.562,160.333
C08711=1019.252,402.752,342.256,173.172,50.561,160.335
C08712=1019.263,402.998,342.211,173.183,50.562,160.337
C08713=1019.273,403.244,342.167,173.195,50.562,160.339
C08714=1019.283,403.489,342.122,173.207,50.562,160.341
C08715=1019.293,403.736,342.077,173.219,50.562,160.343
C08716=1019.304,403.981,342.032,173.232,50.563,160.346
C08717=1019.314,404.226,341.986,173.243,50.563,160.348
C08718=1019.324,404.472,341.942,173.255,50.563,160.350
C08719=1019.334,404.718,341.896,173.268,50.563,160.352
C08720=1019.345,404.963,341.852,173.279,50.564,160.354
C08721=1019.355,405.209,341.806,173.292,50.563,160.356
C08722=1019.365,405.454,341.761,173.305,50.564,160.359
C08723=1019.375,405.701,341.716,173.317,50.564,160.361
C08724=1019.386,405.945,341.671,173.330,50.564,160.363
C08725=1019.396,406.191,341.626,173.341,50.565,160.365
C08726=1019.407,406.438,341.581,173.354,50.565,160.367
C08727=1019.417,406.682,341.535,173.366,50.566,160.370
C08728=1019.428,406.928,341.490,173.379,50.566,160.372
C08729=1019.438,407.174,341.445,173.391,50.566,160.374
C08730=1019.449,407.420,341.399,173.404,50.567,160.377
C08731=1019.459,407.665,341.354,173.417,50.567,160.379
C08732=1019.470,407.910,341.309,173.429,50.567,160.381
C08733=1019.481,408.156,341.263,173.442,50.568,160.384
C08734=1019.491,408.402,341.217,173.455,50.568,160.386
C08735=1019.502,408.648,341.172,173.467,50.568,160.388
C08736=1019.512,408.893,341.126,173.480,50.569,160.391
C08737=1019.523,409.139,341.080,173.493,50.569,160.393
C08738=1019.534,409.385,341.034,173.506,50.570,160.395
C08739=1019.544,409.630,340.988,173.518,50.570,160.398
C08740=1019.555,409.875,340.942,173.532,50.571,160.400
C08741=1019.566,410.121,340.896,173.544,50.572,160.403
C08742=1019.576,410.366,340.850,173.557,50.572,160.405
C08743=1019.587,410.612,340.804,173.570,50.573,160.407
C08744=1019.598,410.857,340.757,173.583,50.574,160.410
C08745=1019.608,411.103,340.711,173.596,50.574,160.412
C08746=1019.618,411.348,340.665,173.609,50.575,160.415
C08747=1019.629,411.593,340.618,173.622,50.576,160.417
C08748=1019.641,411.840,340.572,173.636,50.577,160.420
C08749=1019.651,412.082,340.526,173.648,50.577,160.422
C08750=1019.662,412.326,340.480,173.661,50.578,160.425
C08751=1019.672,412.569,340.434,173.674,50.579,160.427
C08752=1019.684,412.812,340.387,173.688,50.579,160.430
C08753=1019.695,413.056,340.342,173.701,50.580,160.432
C08754=1019.706,413.299,340.296,173.714,50.581,160.435
C08755=1019.716,413.543,340.249,173.727,50.582,160.437
C08756=1019.728,413.786,340.202,173.741,50.582,160.440
C08757=1019.738,414.031,340.156,173.754,50.583,160.442
C08758=1019.749,414.276,340.110,173.767,50.584,160.445
C08759=1019.761,414.522,340.063,173.781,50.584,160.447
C08760=1019.772,414.767,340.016,173.794,50.585,160.450
C08761=1019.783,415.013,339.969,173.809,50.586,160.453
C08762=1019.793,415.258,339.922,173.822,50.587,160.455
C08763=1019.805,415.503,339.874,173.836,50.588,160.458
C08764=1019.816,415.748,339.828,173.849,50.589,160.460
C08765=1019.827,415.994,339.780,173.863,50.590,160.463
C08766=1019.839,416.239,339.732,173.877,50.591,160.466
C08767=1019.849,416.484,339.685,173.891,50.592,160.469
C08768=1019.861,416.730,339.638,173.905,50.593,160.471
C08769=1019.872,416.975,339.590,173.918,50.594,160.474
C08770=1019.883,417.220,339.543,173.933,50.595,160.477
C08771=1019.894,417.465,339.496,173.947,50.596,160.480
C08772=1019.906,417.711,339.448,173.961,50.597,160.482
C08773=1019.917,417.957,339.400,173.975,50.598,160.485
C08774=1019.928,418.201,339.353,173.989,50.599,160.488
C08775=1019.940,418.446,339.305,174.003,50.600,160.491
C08776=1019.951,418.691,339.257,174.017,50.601,160.493
C08777=1019.963,418.937,339.210,174.031,50.602,160.496
C08778=1019.975,419.182,339.162,174.046,50.603,160.499
C08779=1019.986,419.427,339.114,174.060,50.604,160.502
C08780=1019.998,419.672,339.066,174.074,50.605,160.505
C08781=1020.009,419.917,339.019,174.089,50.606,160.508
C08782=1020.020,420.163,338.970,174.103,50.608,160.510
C08783=1020.032,420.408,338.923,174.118,50.609,160.513
C08784=1020.044,420.652,338.874,174.133,50.610,160.516
C08785=1020.056,420.898,338.826,174.147,50.611,160.519
C08786=1020.067,421.143,338.778,174.162,50.612,160.522
C08787=1020.078,421.388,338.730,174.176,50.614,160.525
C08788=1020.091,421.633,338.681,174.191,50.615,160.528
C08789=1020.102,421.879,338.633,174.205,50.616,160.531
C08790=1020.114,422.123,338.584,174.220,50.618,160.534
C08791=1020.126,422.368,338.535,174.235,50.619,160.537
C08792=1020.138,422.613,338.488,174.249,50.620,160.540
C08793=1019.763,420.642,338.538,174.118,50.680,160.534
C08794=1019.751,420.397,338.586,174.104,50.679,160.531
C08795=1019.740,420.152,338.634,174.089,50.678,160.528
C08796=1019.728,419.907,338.682,174.075,50.676,160.525
C08797=1019.717,419.661,338.730,174.060,50.676,160.522
C08798=1019.705,419.416,338.778,174.046,50.675,160.520
C08799=1019.693,419.171,338.826,174.031,50.674,160.517
C08800=1019.682,418.926,338.874,174.017,50.673,160.514
C08801=1019.670,418.681,338.922,174.003,50.672,160.511
C08802=1019.658,418.436,338.969,173.988,50.671,160.508
C08803=1019.648,418.190,339.016,173.975,50.670,160.506
C08804=1019.636,417.945,339.064,173.961,50.669,160.503
C08805=1019.624,417.700,339.112,173.946,50.668,160.500
C08806=1019.614,417.454,339.159,173.932,50.667,160.497
C08807=1019.602,417.210,339.207,173.918,50.666,160.495
C08808=1019.591,416.964,339.254,173.905,50.665,160.492
C08809=1019.580,416.719,339.302,173.890,50.665,160.489
C08810=1019.568,416.473,339.349,173.876,50.663,160.486
C08811=1019.557,416.229,339.396,173.863,50.662,160.484
C08812=1019.546,415.983,339.444,173.849,50.662,160.481
C08813=1019.535,415.738,339.491,173.835,50.661,160.478
C08814=1019.523,415.493,339.538,173.821,50.660,160.476
C08815=1019.513,415.248,339.586,173.807,50.660,160.473
C08816=1019.502,415.002,339.633,173.794,50.659,160.471
C08817=1019.491,414.757,339.679,173.780,50.658,160.468
C08818=1019.479,414.511,339.726,173.767,50.657,160.465
C08819=1019.468,414.266,339.773,173.753,50.656,160.463
C08820=1019.457,414.021,339.820,173.740,50.656,160.460
C08821=1019.447,413.775,339.867,173.726,50.655,160.458
C08822=1019.436,413.545,339.911,173.713,50.655,160.455
C08823=1019.426,413.315,339.954,173.700,50.654,160.453
C08824=1019.416,413.085,339.998,173.688,50.653,160.450
C08825=1019.405,412.855,340.042,173.676,50.653,160.448
C08826=1019.395,412.625,340.085,173.663,50.652,160.446
C08827=1019.385,412.394,340.128,173.650,50.652,160.443
C08828=1019.375,412.164,340.172,173.638,50.651,160.441
C08829=1019.364,411.934,340.216,173.626,50.650,160.439
C08830=1019.353,411.689,340.262,173.613,50.650,160.436
C08831=1019.343,411.443,340.308,173.599,50.650,160.434
C08832=1019.332,411.197,340.354,173.586,50.649,160.431
C08833=1019.321,410.952,340.401,173.573,50.648,160.429
C08834=1019.310,410.706,340.447,173.560,50.648,160.427
C08835=1019.299,410.461,340.493,173.548,50.648,160.424
C08836=1019.288,410.216,340.539,173.534,50.647,160.422
C08837=1019.278,409.970,340.586,173.521,50.646,160.419
C08838=1019.268,409.724,340.632,173.508,50.646,160.417
C08839=1019.257,409.478,340.678,173.495,50.646,160.415
C08840=1019.247,409.233,340.724,173.483,50.645,160.412
C08841=1019.237,408.988,340.769,173.470,50.645,160.410
C08842=1019.226,408.742,340.815,173.457,50.644,160.407
C08843=1019.215,408.497,340.861,173.444,50.644,160.405
C08844=1019.204,408.252,340.906,173.431,50.644,160.403
C08845=1019.194,408.005,340.951,173.418,50.644,160.401
C08846=1019.183,407.760,340.997,173.406,50.643,160.398
C08847=1019.172,407.514,341.043,173.393,50.643,160.396
C08848=1019.162,407.268,341.088,173.381,50.643,160.394
C08849=1019.151,407.023,341.133,173.368,50.642,160.391
C08850=1019.141,406.778,341.179,173.355,50.642,160.389
C08851=1019.130,406.532,341.224,173.343,50.642,160.387
C08852=1019.121,406.286,341.269,173.331,50.642,160.385
C08853=1019.109,406.041,341.315,173.319,50.641,160.382
C08854=1019.099,405.795,341.360,173.306,50.641,160.380
C08855=1019.089,405.550,341.405,173.294,50.641,160.378
C08856=1019.079,405.303,341.451,173.281,50.641,160.376
C08857=1019.068,405.058,341.495,173.269,50.641,160.374
C08858=1019.058,404.813,341.541,173.256,50.641,160.371
C08859=1019.047,404.566,341.586,173.245,50.640,160.369
C08860=1019.038,404.321,341.631,173.232,50.640,160.367
C08861=1019.027,404.076,341.675,173.220,50.640,160.365
C08862=1019.017,403.829,341.720,173.208,50.640,160.363
C08863=1019.007,403.584,341.765,173.196,50.640,160.361
C08864=1018.997,403.338,341.810,173.184,50.640,160.358
C08865=1018.986,403.093,341.854,173.172,50.640,160.356
C08866=1018.977,402.847,341.899,173.159,50.640,160.354
C08867=1018.966,402.601,341.944,173.148,50.640,160.352
C08868=1018.957,402.355,341.989,173.136,50.640,160.350
C08869=1018.946,402.110,342.033,173.124,50.640,160.348
C08870=1018.936,401.865,342.078,173.112,50.640,160.346
C08871=1018.926,401.618,342.123,173.100,50.640,160.344
C08872=1018.917,401.372,342.168,173.088,50.640,160.342
C08873=1018.906,401.127,342.212,173.076,50.640,160.339
C08874=1018.897,400.881,342.256,173.065,50.640,160.338
C08875=1018.887,400.635,342.301,173.053,50.640,160.335
C08876=1018.878,400.389,342.345,173.041,50.640,160.333
C08877=1018.867,400.143,342.389,173.029,50.640,160.331
C08878=1018.857,399.897,342.434,173.018,50.640,160.329
C08879=1018.847,399.652,342.478,173.006,50.641,160.327
C08880=1018.837,399.406,342.522,172.995,50.640,160.325
C08881=1018.827,399.160,342.565,172.983,50.641,160.323
C08882=1018.817,398.915,342.610,172.971,50.641,160.321
C08883=1018.808,398.668,342.654,172.959,50.641,160.319
C08884=1018.798,398.423,342.698,172.948,50.642,160.318
C08885=1018.788,398.176,342.742,172.936,50.642,160.315
C08886=1018.776,397.843,342.801,172.921,50.642,160.313
C08887=1018.762,397.508,342.861,172.906,50.642,160.310
C08888=1018.749,397.175,342.920,172.890,50.643,160.308
C08889=1018.736,396.841,342.979,172.875,50.643,160.305
C08890=1018.726,396.595,343.023,172.863,50.644,160.303
C08891=1018.716,396.349,343.066,172.852,50.644,160.301
C08892=1018.706,396.103,343.110,172.841,50.644,160.300
C08893=1018.696,395.857,343.153,172.829,50.645,160.298
C08894=1018.687,395.611,343.197,172.818,50.645,160.296
C08895=1018.677,395.366,343.240,172.807,50.645,160.294
C08896=1018.668,395.119,343.283,172.796,50.646,160.292
C08897=1018.658,394.873,343.327,172.784,50.646,160.290
C08898=1018.649,394.627,343.370,172.773,50.646,160.288
C08899=1018.639,394.381,343.413,172.763,50.647,160.287
C08900=1018.630,394.135,343.457,172.752,50.648,160.285
C08901=1018.620,393.890,343.500,172.741,50.648,160.283
C08902=1018.610,393.643,343.543,172.729,50.648,160.281
C08903=1018.601,393.397,343.587,172.718,50.649,160.279
C08904=1018.592,393.151,343.629,172.707,50.649,160.278
C08905=1018.582,392.905,343.672,172.696,50.650,160.276
C08906=1018.573,392.659,343.716,172.686,50.651,160.274
C08907=1018.563,392.413,343.759,172.675,50.651,160.272
C08908=1018.554,392.167,343.801,172.664,50.652,160.271
C08909=1018.545,391.920,343.844,172.653,50.652,160.269
C08910=1018.536,391.675,343.887,172.643,50.653,160.267
C08911=1018.526,391.428,343.930,172.631,50.653,160.265
C08912=1018.517,391.182,343.972,172.620,50.654,160.264
C08913=1018.507,390.937,344.014,172.610,50.655,160.262
C08914=1018.497,390.690,344.057,172.599,50.655,160.260
C08915=1018.489,390.444,344.100,172.588,50.656,160.258
C08916=1018.479,390.198,344.143,172.578,50.657,160.257
C08917=1018.470,389.952,344.185,172.567,50.658,160.255
C08918=1018.461,389.706,344.227,172.556,50.658,160.253
C08919=1018.452,389.460,344.270,172.546,50.659,160.252
C08920=1018.443,389.213,344.313,172.536,50.659,160.250
C08921=1018.434,388.967,344.355,172.525,50.660,160.249
C08922=1018.424,388.721,344.397,172.515,50.661,160.247
C08923=1018.415,388.475,344.440,172.504,50.662,160.245
C08924=1018.406,388.228,344.482,172.494,50.663,160.244
C08925=1018.396,387.982,344.524,172.483,50.663,160.242
C08926=1018.387,387.736,344.566,172.473,50.664,160.240
C08927=1018.378,387.490,344.608,172.462,50.665,160.239
C08928=1018.369,387.244,344.650,172.451,50.666,160.237
C08929=1018.360,386.998,344.692,172.442,50.666,160.236
C08930=1018.351,386.751,344.735,172.432,50.668,160.234
C08931=1018.342,386.505,344.776,172.421,50.669,160.233
C08932=1018.333,386.258,344.818,172.411,50.669,160.231
C08933=1018.324,386.012,344.861,172.400,50.670,160.229
C08934=1018.315,385.766,344.903,172.390,50.672,160.228
C08935=1018.306,385.520,344.944,172.380,50.672,160.226
C08936=1018.297,385.273,344.986,172.370,50.673,160.225
C08937=1018.288,385.027,345.028,172.360,50.674,160.223
C08938=1018.279,384.781,345.069,172.349,50.675,160.222
C08939=1018.270,384.535,345.111,172.340,50.676,160.220
C08940=1018.261,384.288,345.152,172.329,50.677,160.219
C08941=1018.252,384.042,345.194,172.319,50.678,160.217
C08942=1018.242,383.796,345.235,172.308,50.679,160.216
C08943=1018.234,383.549,345.276,172.299,50.680,160.214
C08944=1018.225,383.303,345.318,172.289,50.682,160.213
C08945=1018.216,383.057,345.359,172.279,50.682,160.211
C08946=1018.205,382.760,345.409,172.267,50.684,160.209
C08947=1018.194,382.463,345.458,172.254,50.685,160.208
C08948=1018.184,382.167,345.508,172.243,50.686,160.206
C08949=1018.173,381.871,345.557,172.231,50.688,160.204
C08950=1018.164,381.625,345.599,172.221,50.689,160.203
C08951=1018.156,381.378,345.640,172.211,50.690,160.201
C08952=1018.147,381.132,345.682,172.202,50.691,160.200
C08953=1018.138,380.885,345.723,172.192,50.693,160.199
C08954=1018.129,380.639,345.763,172.181,50.694,160.197
C08955=1018.120,380.392,345.804,172.172,50.695,160.196
C08956=1018.112,380.145,345.845,172.162,50.697,160.194
C08957=1018.103,379.900,345.887,172.153,50.698,160.193
C08958=1018.094,379.653,345.927,172.143,50.699,160.192
C08959=1018.086,379.407,345.968,172.133,50.700,160.190
C08960=1018.077,379.160,346.009,172.123,50.701,160.189
C08961=1018.069,378.913,346.050,172.114,50.703,160.188
C08962=1018.060,378.667,346.090,172.104,50.704,160.186
C08963=1018.051,378.420,346.131,172.095,50.705,160.185
C08964=1018.043,378.174,346.172,172.085,50.707,160.184
C08965=1018.034,377.927,346.213,172.076,50.708,160.182
C08966=1018.026,377.681,346.253,172.066,50.709,160.181
C08967=1018.017,377.434,346.294,172.056,50.710,160.180
C08968=1018.009,377.188,346.335,172.047,50.712,160.178
C08969=1018.001,376.942,346.375,172.037,50.714,160.177
C08970=1017.992,376.695,346.416,172.027,50.715,160.176
C08971=1017.984,376.449,346.456,172.018,50.716,160.174
C08972=1017.975,376.202,346.497,172.009,50.718,160.173
C08973=1017.967,375.955,346.538,171.999,50.719,160.172
C08974=1017.959,375.709,346.579,171.990,50.721,160.171
C08975=1017.950,375.462,346.618,171.980,50.722,160.169
C08976=1017.941,375.216,346.658,171.971,50.724,160.168
C08977=1017.933,374.970,346.699,171.962,50.725,160.167
C08978=1017.924,374.722,346.739,171.952,50.727,160.166
C08979=1017.916,374.476,346.779,171.944,50.728,160.164
C08980=1017.908,374.229,346.819,171.933,50.730,160.163
C08981=1017.899,373.982,346.860,171.925,50.731,160.162
C08982=1017.890,373.736,346.899,171.916,50.733,160.161
C08983=1017.882,373.490,346.939,171.906,50.735,160.160
C08984=1017.874,373.243,346.979,171.897,50.736,160.158
C08985=1017.866,372.996,347.018,171.888,50.738,160.157
C08986=1017.857,372.749,347.059,171.878,50.740,160.156
C08987=1017.848,372.503,347.099,171.870,50.741,160.155
C08988=1017.841,372.256,347.139,171.861,50.743,160.154
C08989=1017.832,372.010,347.179,171.851,50.744,160.152
C08990=1017.824,371.763,347.218,171.842,50.746,160.151
C08991=1017.816,371.516,347.258,171.833,50.748,160.150
C08992=1017.807,371.270,347.297,171.824,50.749,160.149
C08993=1017.799,371.022,347.337,171.814,50.751,160.148
C08994=1017.791,370.776,347.377,171.806,50.753,160.146
C08995=1017.783,370.529,347.417,171.797,50.755,160.145
C08996=1017.774,370.283,347.457,171.788,50.756,160.144
C08997=1017.766,370.036,347.496,171.778,50.758,160.143
C08998=1017.758,369.789,347.536,171.769,50.760,160.142
C08999=1017.749,369.543,347.575,171.761,50.762,160.141
C09000=1017.742,369.296,347.615,171.752,50.764,160.140
C09001=1017.734,369.049,347.653,171.744,50.765,160.139
C09002=1017.726,368.803,347.693,171.735,50.767,160.138
C09003=1017.718,368.556,347.733,171.725,50.769,160.136
C09004=1017.710,368.309,347.772,171.717,50.771,160.135
C09005=1017.702,368.062,347.812,171.708,50.773,160.134
C09006=1017.693,367.788,347.855,171.698,50.775,160.133
C09007=1017.684,367.514,347.899,171.688,50.777,160.132
C09008=1017.675,367.240,347.942,171.678,50.779,160.131
C09009=1017.666,366.967,347.986,171.669,50.782,160.130
C09010=1017.658,366.719,348.025,171.660,50.783,160.129
C09011=1017.649,366.473,348.064,171.651,50.785,160.127
C09012=1017.641,366.226,348.102,171.642,50.787,160.126
C09013=1017.633,365.979,348.142,171.634,50.790,160.125
C09014=1017.625,365.733,348.180,171.625,50.791,160.124
C09015=1017.617,365.485,348.219,171.616,50.794,160.123
C09016=1017.609,365.239,348.258,171.608,50.795,160.122
C09017=1017.601,364.991,348.297,171.599,50.797,160.121
C09018=1017.594,364.745,348.335,171.591,50.800,160.120
C09019=1017.585,364.498,348.375,171.582,50.801,160.119
C09020=1017.577,364.251,348.413,171.574,50.804,160.118
C09021=1017.570,364.004,348.452,171.564,50.806,160.117
C09022=1017.561,363.757,348.490,171.555,50.808,160.116
C09023=1017.553,363.511,348.530,171.547,50.810,160.115
C09024=1017.545,363.264,348.568,171.539,50.812,160.114
C09025=1017.537,363.017,348.606,171.530,50.815,160.114
C09026=1017.530,362.770,348.645,171.522,50.817,160.113
C09027=1017.522,362.523,348.683,171.513,50.818,160.111
C09028=1017.513,362.276,348.722,171.505,50.821,160.111
C09029=1017.507,362.029,348.761,171.496,50.823,160.110
C09030=1017.498,361.782,348.799,171.488,50.825,160.109
C09031=1017.491,361.535,348.838,171.479,50.828,160.108
C09032=1017.483,361.288,348.876,171.471,50.830,160.107
C09033=1017.475,361.042,348.914,171.463,50.832,160.106
C09034=1017.468,360.795,348.953,171.454,50.834,160.105
C09035=1017.459,360.548,348.991,171.446,50.837,160.104
C09036=1017.452,360.301,349.029,171.437,50.839,160.103
C09037=1017.444,360.053,349.067,171.429,50.841,160.102
C09038=1017.437,359.807,349.106,171.421,50.843,160.101
C09039=1017.428,359.560,349.144,171.412,50.846,160.100
C09040=1017.421,359.313,349.182,171.405,50.847,160.100
C09041=1017.414,359.066,349.220,171.397,50.850,160.099
C09042=1017.405,358.819,349.259,171.388,50.853,160.098
C09043=1017.398,358.572,349.297,171.380,50.855,160.097
C09044=1017.391,358.325,349.334,171.372,50.857,160.096
C09045=1017.383,358.078,349.373,171.364,50.860,160.095
C09046=1017.375,357.831,349.410,171.355,50.862,160.095
C09047=1017.367,357.585,349.448,171.347,50.864,160.094
C09048=1017.359,357.337,349.486,171.339,50.867,160.093
C09049=1017.352,357.090,349.524,171.330,50.870,160.092
C09050=1017.344,356.843,349.562,171.322,50.872,160.091
C09051=1017.337,356.596,349.599,171.314,50.875,160.090
C09052=1017.329,356.349,349.637,171.306,50.877,160.089
C09053=1017.321,356.102,349.675,171.298,50.880,160.089
C09054=1017.314,355.855,349.712,171.290,50.882,160.088
C09055=1017.306,355.608,349.750,171.282,50.885,160.087
C09056=1017.298,355.361,349.787,171.274,50.887,160.086
C09057=1017.291,355.113,349.825,171.266,50.890,160.086
C09058=1017.283,354.867,349.863,171.258,50.893,160.085
C09059=1017.276,354.619,349.901,171.249,50.895,160.084
C09060=1017.268,354.373,349.937,171.241,50.898,160.083
C09061=1017.261,354.125,349.975,171.234,50.900,160.083
C09062=1017.253,353.878,350.012,171.226,50.902,160.082
C09063=1017.246,353.631,350.050,171.218,50.905,160.081
C09064=1017.238,353.384,350.087,171.210,50.908,160.080
C09065=1017.231,353.137,350.124,171.202,50.911,160.080
C09066=1017.222,352.870,350.165,171.194,50.913,160.079
C09067=1017.214,352.604,350.205,171.185,50.917,160.078
C09068=1017.206,352.338,350.245,171.177,50.919,160.077
C09069=1017.198,352.071,350.285,171.168,50.923,160.076
C09070=1017.190,351.825,350.322,171.161,50.925,160.076
C09071=1017.183,351.577,350.359,171.153,50.928,160.075
C09072=1017.175,351.330,350.396,171.145,50.931,160.074
C09073=1017.168,351.083,350.433,171.137,50.934,160.074
C09074=1017.160,350.836,350.470,171.129,50.937,160.073
C09075=1017.153,350.588,350.507,171.121,50.940,160.072
C09076=1017.146,350.341,350.544,171.114,50.942,160.071
C09077=1017.138,350.094,350.581,171.106,50.945,160.071
C09078=1017.131,349.847,350.618,171.098,50.948,160.070
C09079=1017.124,349.600,350.655,171.090,50.951,160.069
C09080=1017.117,349.353,350.692,171.083,50.953,160.069
C09081=1017.109,349.106,350.729,171.075,50.956,160.068
C09082=1017.102,348.858,350.765,171.067,50.959,160.067
C09083=1017.094,348.611,350.802,171.059,50.962,160.067
C09084=1017.087,348.363,350.839,171.052,50.965,160.066
C09085=1017.080,348.117,350.876,171.044,50.968,160.065
C09086=1017.073,347.870,350.912,171.036,50.971,160.065
C09087=1017.066,347.622,350.949,171.028,50.974,160.064
